LIN {X -0.219,Y -497.782,Z 714.673,A 0.000,B 0.000,C 90.000,E1 337.230} C_DIS
LIN {X 0.009,Y -502.291,Z 714.671,A 0.000,B 0.000,C 90.000,E1 336.794} C_DIS
LIN {X -0.050,Y -508.805,Z 714.668,A 0.000,B 0.000,C 90.000,E1 336.305} C_DIS
LIN {X 0.103,Y -528.863,Z 714.661,A 0.000,B 0.000,C 90.000,E1 334.973} C_DIS
LIN {X -0.127,Y -535.110,Z 714.659,A 0.000,B 0.000,C 90.000,E1 334.588} C_DIS
LIN {X -0.009,Y -541.078,Z 714.656,A 0.000,B 0.000,C 90.000,E1 334.152} C_DIS
LIN {X 0.145,Y -548.131,Z 714.653,A 0.000,B 0.000,C 90.000,E1 333.589} C_DIS
LIN {X -0.065,Y -552.381,Z 714.651,A 0.000,B 0.000,C 90.000,E1 333.256} C_DIS
LIN {X -0.107,Y -557.683,Z 714.649,A 0.000,B 0.000,C 90.000,E1 332.794} C_DIS
LIN {X 0.163,Y -562.857,Z 714.646,A 0.000,B 0.000,C 90.000,E1 332.281} C_DIS
LIN {X 0.153,Y -568.016,Z 714.643,A 0.000,B 0.000,C 90.000,E1 331.769} C_DIS
LIN {X -0.083,Y -574.316,Z 714.640,A 0.000,B 0.000,C 90.000,E1 331.129} C_DIS
LIN {X -0.285,Y -582.771,Z 714.634,A 0.000,B 0.000,C 90.000,E1 330.205} C_DIS
LIN {X -0.328,Y -588.752,Z 714.631,A 0.000,B 0.000,C 90.000,E1 329.537} C_DIS
LIN {X -0.316,Y -594.337,Z 714.627,A 0.000,B 0.000,C 90.000,E1 328.869} C_DIS
LIN {X -0.028,Y -601.884,Z 714.622,A 0.000,B 0.000,C 90.000,E1 327.916} C_DIS
LIN {X 0.100,Y -607.002,Z 714.618,A 0.000,B 0.000,C 90.000,E1 327.248} C_DIS
LIN {X -0.242,Y -611.865,Z 714.615,A 0.000,B 0.000,C 90.000,E1 326.628} C_DIS
LIN {X -0.035,Y -616.443,Z 714.611,A 0.000,B 0.000,C 90.000,E1 325.960} C_DIS
LIN {X 0.030,Y -621.689,Z 714.607,A 0.000,B 0.000,C 90.000,E1 325.182} C_DIS
LIN {X -0.304,Y -628.155,Z 714.601,A 0.000,B 0.000,C 90.000,E1 324.196} C_DIS
LIN {X 0.253,Y -634.206,Z 714.595,A 0.000,B 0.000,C 90.000,E1 323.130} C_DIS
LIN {X -0.001,Y -639.822,Z 714.590,A 0.000,B 0.000,C 90.000,E1 322.145} C_DIS
LIN {X 0.200,Y -644.512,Z 714.585,A 0.000,B 0.000,C 90.000,E1 321.251} C_DIS
LIN {X -0.021,Y -650.301,Z 714.579,A 0.000,B 0.000,C 90.000,E1 320.150} C_DIS
LIN {X 0.256,Y -655.679,Z 714.572,A 0.000,B 0.000,C 90.000,E1 319.013} C_DIS
LIN {X -0.332,Y -660.202,Z 714.567,A 0.000,B 0.000,C 90.000,E1 318.081} C_DIS
LIN {X 0.074,Y -664.376,Z 714.562,A 0.000,B 0.000,C 90.000,E1 317.067} C_DIS
LIN {X 0.054,Y -667.312,Z 714.557,A 0.000,B 0.000,C 90.000,E1 316.338} C_DIS
LIN {X 0.086,Y -670.924,Z 714.552,A 0.000,B 0.000,C 90.000,E1 315.364} C_DIS
LIN {X -0.303,Y -675.162,Z 714.545,A 0.000,B 0.000,C 90.000,E1 314.190} C_DIS
LIN {X -0.155,Y -679.089,Z 714.539,A 0.000,B 0.000,C 90.000,E1 312.975} C_DIS
LIN {X 0.091,Y -682.786,Z 714.532,A 0.000,B 0.000,C 90.000,E1 311.757} C_DIS
LIN {X -0.168,Y -685.479,Z 714.527,A 0.000,B 0.000,C 90.000,E1 310.825} C_DIS
LIN {X 0.124,Y -688.027,Z 714.521,A 0.000,B 0.000,C 90.000,E1 309.850} C_DIS
LIN {X 0.013,Y -690.186,Z 714.516,A 0.000,B 0.000,C 90.000,E1 308.910} C_DIS
LIN {X 0.303,Y -691.640,Z 714.512,A 0.000,B 0.000,C 90.000,E1 308.177} C_DIS
LIN {X 0.247,Y -693.299,Z 714.507,A 0.000,B 0.000,C 90.000,E1 307.237} C_DIS
LIN {X -0.145,Y -695.119,Z 714.500,A 0.000,B 0.000,C 90.000,E1 306.091} C_DIS
LIN {X -0.169,Y -696.354,Z 714.495,A 0.000,B 0.000,C 90.000,E1 305.152} C_DIS
LIN {X -0.353,Y -697.682,Z 714.489,A 0.000,B 0.000,C 90.000,E1 303.992} C_DIS
LIN {X 0.174,Y -698.364,Z 714.485,A 0.000,B 0.000,C 90.000,E1 303.245} C_DIS
LIN {X 0.321,Y -699.714,Z 714.476,A 0.000,B 0.000,C 90.000,E1 301.592} C_DIS
LIN {X 0.166,Y -700.447,Z 714.471,A 0.000,B 0.000,C 90.000,E1 300.669} C_DIS
LIN {X -0.244,Y -700.786,Z 714.467,A 0.000,B 0.000,C 90.000,E1 300.001} C_DIS
LIN {X -0.180,Y -701.290,Z 714.458,A 0.000,B 0.000,C 90.000,E1 298.359} C_DIS
LIN {X -0.160,Y -701.935,Z 714.447,A 0.000,B 0.000,C 90.000,E1 296.488} C_DIS
LIN {X 0.016,Y -702.412,Z 714.442,A 0.000,B 0.000,C 90.000,E1 295.540} C_DIS
LIN {X -0.061,Y -702.510,Z 714.439,A 0.000,B 0.000,C 90.000,E1 295.079} C_DIS
LIN {X 0.201,Y -701.996,Z 714.437,A 0.000,B 0.000,C 90.000,E1 294.591} C_DIS
LIN {X -0.160,Y -701.436,Z 714.435,A 0.000,B 0.000,C 90.000,E1 294.387} C_DIS
LIN {X 0.101,Y -699.381,Z 714.433,A 0.000,B 0.000,C 90.000,E1 293.898} C_DIS
LIN {X 0.237,Y -698.741,Z 714.432,A 0.000,B 0.000,C 90.000,E1 293.770} C_DIS
LIN {X -0.269,Y -697.777,Z 714.432,A 0.000,B 0.000,C 90.000,E1 293.695} C_DIS
LIN {X -0.138,Y -696.354,Z 714.431,A 0.000,B 0.000,C 90.000,E1 293.567} C_DIS
LIN {X 0.001,Y -690.082,Z 714.429,A 0.000,B 0.000,C 90.000,E1 293.153} C_DIS
LIN {X -0.210,Y -687.788,Z 714.428,A 0.000,B 0.000,C 90.000,E1 293.078} C_DIS
LIN {X -0.113,Y -685.753,Z 714.428,A 0.000,B 0.000,C 90.000,E1 293.003} C_DIS
LIN {X -0.153,Y -677.503,Z 714.427,A 0.000,B 0.000,C 90.000,E1 292.823} C_DIS
LIN {X -0.057,Y -659.849,Z 714.426,A 0.000,B 0.000,C 90.000,E1 292.589} C_DIS
LIN {X -0.180,Y -646.131,Z 714.424,A 0.000,B 0.000,C 90.000,E1 292.386} C_DIS
LIN {X -0.277,Y -636.241,Z 714.423,A 0.000,B 0.000,C 90.000,E1 292.206} C_DIS
LIN {X -0.263,Y -622.792,Z 714.422,A 0.000,B 0.000,C 90.000,E1 291.897} C_DIS
LIN {X -0.150,Y -602.290,Z 714.419,A 0.000,B 0.000,C 90.000,E1 291.334} C_DIS
LIN {X 0.095,Y -574.338,Z 714.414,A 0.000,B 0.000,C 90.000,E1 290.482} C_DIS
LIN {X -0.073,Y -567.828,Z 714.413,A 0.000,B 0.000,C 90.000,E1 290.301} C_DIS
LIN {X 0.069,Y -561.417,Z 714.412,A 0.000,B 0.000,C 90.000,E1 290.066} C_DIS
LIN {X -0.026,Y -559.588,Z 714.411,A 0.000,B 0.000,C 90.000,E1 289.993} C_DIS
LIN {X 0.055,Y -556.344,Z 714.410,A 0.000,B 0.000,C 90.000,E1 289.758} C_DIS
LIN {X 0.001,Y -556.275,Z 714.410,A 0.000,B 0.000,C 90.000,E1 289.758} C_DIS
LIN {X -0.250,Y -555.291,Z 714.409,A 0.000,B 0.000,C 90.000,E1 289.577} C_DIS
LIN {X 0.256,Y -554.824,Z 714.407,A 0.000,B 0.000,C 90.000,E1 289.141} C_DIS
LIN {X -0.162,Y -554.077,Z 714.397,A 0.000,B 0.000,C 90.000,E1 287.511} C_DIS
LIN {X -0.230,Y -553.446,Z 714.388,A 0.000,B 0.000,C 90.000,E1 285.843} C_DIS
LIN {X -0.194,Y -552.769,Z 714.377,A 0.000,B 0.000,C 90.000,E1 283.883} C_DIS
LIN {X -0.134,Y -552.316,Z 714.369,A 0.000,B 0.000,C 90.000,E1 282.479} C_DIS
LIN {X -0.075,Y -551.743,Z 714.362,A 0.000,B 0.000,C 90.000,E1 281.074} C_DIS
LIN {X 0.078,Y -550.988,Z 714.352,A 0.000,B 0.000,C 90.000,E1 279.378} C_DIS
LIN {X 0.134,Y -550.123,Z 714.341,A 0.000,B 0.000,C 90.000,E1 277.409} C_DIS
LIN {X 0.270,Y -549.218,Z 714.326,A 0.000,B 0.000,C 90.000,E1 274.588} C_DIS
LIN {X -0.005,Y -548.880,Z 714.318,A 0.000,B 0.000,C 90.000,E1 273.212} C_DIS
LIN {X -0.212,Y -548.201,Z 714.309,A 0.000,B 0.000,C 90.000,E1 271.547} C_DIS
LIN {X 0.029,Y -547.571,Z 714.301,A 0.000,B 0.000,C 90.000,E1 270.115} C_DIS
LIN {X -0.243,Y -546.555,Z 714.291,A 0.000,B 0.000,C 90.000,E1 268.453} C_DIS
LIN {X 0.080,Y -545.356,Z 714.280,A 0.000,B 0.000,C 90.000,E1 266.445} C_DIS
LIN {X -0.226,Y -544.321,Z 714.273,A 0.000,B 0.000,C 90.000,E1 265.065} C_DIS
LIN {X 0.065,Y -543.053,Z 714.263,A 0.000,B 0.000,C 90.000,E1 263.337} C_DIS
LIN {X 0.236,Y -542.050,Z 714.257,A 0.000,B 0.000,C 90.000,E1 262.186} C_DIS
LIN {X 0.077,Y -540.569,Z 714.247,A 0.000,B 0.000,C 90.000,E1 260.500} C_DIS
LIN {X -0.110,Y -539.017,Z 714.238,A 0.000,B 0.000,C 90.000,E1 258.814} C_DIS
LIN {X 0.230,Y -537.809,Z 714.230,A 0.000,B 0.000,C 90.000,E1 257.353} C_DIS
LIN {X -0.268,Y -535.922,Z 714.219,A 0.000,B 0.000,C 90.000,E1 255.408} C_DIS
LIN {X 0.217,Y -534.819,Z 714.212,A 0.000,B 0.000,C 90.000,E1 254.212} C_DIS
LIN {X -0.064,Y -532.775,Z 714.201,A 0.000,B 0.000,C 90.000,E1 252.236} C_DIS
LIN {X 0.061,Y -531.289,Z 714.193,A 0.000,B 0.000,C 90.000,E1 250.786} C_DIS
LIN {X -0.039,Y -529.850,Z 714.187,A 0.000,B 0.000,C 90.000,E1 249.645} C_DIS
LIN {X -0.118,Y -527.448,Z 714.177,A 0.000,B 0.000,C 90.000,E1 247.922} C_DIS
LIN {X -0.215,Y -525.392,Z 714.169,A 0.000,B 0.000,C 90.000,E1 246.485} C_DIS
LIN {X -0.129,Y -523.062,Z 714.161,A 0.000,B 0.000,C 90.000,E1 245.025} C_DIS
LIN {X 0.012,Y -521.122,Z 714.155,A 0.000,B 0.000,C 90.000,E1 243.845} C_DIS
LIN {X 0.112,Y -518.980,Z 714.148,A 0.000,B 0.000,C 90.000,E1 242.666} C_DIS
LIN {X 0.332,Y -515.004,Z 714.137,A 0.000,B 0.000,C 90.000,E1 240.589} C_DIS
LIN {X -0.007,Y -511.908,Z 714.129,A 0.000,B 0.000,C 90.000,E1 239.154} C_DIS
LIN {X 0.022,Y -508.132,Z 714.119,A 0.000,B 0.000,C 90.000,E1 237.375} C_DIS
LIN {X 0.084,Y -505.076,Z 714.111,A 0.000,B 0.000,C 90.000,E1 235.881} C_DIS
LIN {X -0.048,Y -501.706,Z 714.102,A 0.000,B 0.000,C 90.000,E1 234.402} C_DIS
LIN {X 0.005,Y -499.577,Z 714.097,A 0.000,B 0.000,C 90.000,E1 233.497} C_DIS
LIN {X -0.242,Y -498.059,Z 714.094,A 0.000,B 0.000,C 90.000,E1 232.924} C_DIS
LIN {X -0.190,Y -492.612,Z 714.082,A 0.000,B 0.000,C 90.000,E1 230.803} C_DIS
LIN {X 0.028,Y -487.561,Z 714.070,A 0.000,B 0.000,C 90.000,E1 228.647} C_DIS
LIN {X -0.247,Y -484.070,Z 714.062,A 0.000,B 0.000,C 90.000,E1 227.148} C_DIS
LIN {X 0.103,Y -480.666,Z 714.053,A 0.000,B 0.000,C 90.000,E1 225.567} C_DIS
LIN {X -0.063,Y -475.888,Z 714.041,A 0.000,B 0.000,C 90.000,E1 223.419} C_DIS
LIN {X -0.095,Y -471.932,Z 714.031,A 0.000,B 0.000,C 90.000,E1 221.553} C_DIS
LIN {X 0.056,Y -468.580,Z 714.022,A 0.000,B 0.000,C 90.000,E1 219.967} C_DIS
LIN {X 0.135,Y -465.177,Z 714.013,A 0.000,B 0.000,C 90.000,E1 218.382} C_DIS
LIN {X -0.177,Y -459.559,Z 713.999,A 0.000,B 0.000,C 90.000,E1 215.884} C_DIS
LIN {X 0.093,Y -454.588,Z 713.985,A 0.000,B 0.000,C 90.000,E1 213.293} C_DIS
LIN {X 0.197,Y -451.580,Z 713.976,A 0.000,B 0.000,C 90.000,E1 211.671} C_DIS
LIN {X 0.015,Y -448.625,Z 713.967,A 0.000,B 0.000,C 90.000,E1 210.079} C_DIS
LIN {X -0.226,Y -445.600,Z 713.958,A 0.000,B 0.000,C 90.000,E1 208.487} C_DIS
LIN {X 0.047,Y -442.692,Z 713.949,A 0.000,B 0.000,C 90.000,E1 206.821} C_DIS
LIN {X 0.107,Y -439.100,Z 713.938,A 0.000,B 0.000,C 90.000,E1 204.847} C_DIS
LIN {X 0.061,Y -436.090,Z 713.929,A 0.000,B 0.000,C 90.000,E1 203.206} C_DIS
LIN {X 0.049,Y -431.196,Z 713.914,A 0.000,B 0.000,C 90.000,E1 200.556} C_DIS
LIN {X 0.112,Y -428.778,Z 713.907,A 0.000,B 0.000,C 90.000,E1 199.214} C_DIS
LIN {X 0.185,Y -424.473,Z 713.894,A 0.000,B 0.000,C 90.000,E1 196.858} C_DIS
LIN {X -0.111,Y -420.154,Z 713.881,A 0.000,B 0.000,C 90.000,E1 194.537} C_DIS
LIN {X 0.176,Y -415.922,Z 713.867,A 0.000,B 0.000,C 90.000,E1 192.119} C_DIS
LIN {X 0.124,Y -412.367,Z 713.856,A 0.000,B 0.000,C 90.000,E1 190.074} C_DIS
LIN {X -0.083,Y -407.368,Z 713.839,A 0.000,B 0.000,C 90.000,E1 187.004} C_DIS
LIN {X -0.123,Y -404.773,Z 713.829,A 0.000,B 0.000,C 90.000,E1 185.277} C_DIS
LIN {X 0.100,Y -401.334,Z 713.816,A 0.000,B 0.000,C 90.000,E1 182.808} C_DIS
LIN {X 0.032,Y -397.177,Z 713.796,A 0.000,B 0.000,C 90.000,E1 179.312} C_DIS
LIN {X -0.113,Y -394.188,Z 713.779,A 0.000,B 0.000,C 90.000,E1 176.159} C_DIS
LIN {X 0.198,Y -392.236,Z 713.763,A 0.000,B 0.000,C 90.000,E1 173.280} C_DIS
LIN {X -0.130,Y -391.098,Z 713.751,A 0.000,B 0.000,C 90.000,E1 171.197} C_DIS
LIN {X -0.128,Y -389.907,Z 713.733,A 0.000,B 0.000,C 90.000,E1 167.993} C_DIS
LIN {X 0.103,Y -389.112,Z 713.719,A 0.000,B 0.000,C 90.000,E1 165.463} C_DIS
LIN {X 0.064,Y -388.736,Z 713.709,A 0.000,B 0.000,C 90.000,E1 163.685} C_DIS
LIN {X 0.119,Y -388.531,Z 713.700,A 0.000,B 0.000,C 90.000,E1 161.891} C_DIS
LIN {X 0.119,Y -388.413,Z 713.686,A 0.000,B 0.000,C 90.000,E1 159.390} C_DIS
LIN {X 0.101,Y -388.434,Z 713.668,A 0.000,B 0.000,C 90.000,E1 156.177} C_DIS
LIN {X 0.000,Y -388.663,Z 713.654,A 0.000,B 0.000,C 90.000,E1 153.691} C_DIS
LIN {X 0.059,Y -388.912,Z 713.644,A 0.000,B 0.000,C 90.000,E1 151.897} C_DIS
LIN {X 0.061,Y -389.865,Z 713.624,A 0.000,B 0.000,C 90.000,E1 148.329} C_DIS
LIN {X 0.145,Y -393.306,Z 713.596,A 0.000,B 0.000,C 90.000,E1 143.336} C_DIS
LIN {X -0.120,Y -395.537,Z 713.585,A 0.000,B 0.000,C 90.000,E1 141.251} C_DIS
LIN {X 0.067,Y -399.294,Z 713.569,A 0.000,B 0.000,C 90.000,E1 138.405} C_DIS
LIN {X -0.206,Y -401.196,Z 713.563,A 0.000,B 0.000,C 90.000,E1 137.391} C_DIS
LIN {X 0.178,Y -402.104,Z 713.561,A 0.000,B 0.000,C 90.000,E1 136.986} C_DIS
LIN {X -0.061,Y -403.913,Z 713.558,A 0.000,B 0.000,C 90.000,E1 136.458} C_DIS
LIN {X 0.254,Y -406.545,Z 713.555,A 0.000,B 0.000,C 90.000,E1 135.891} C_DIS
LIN {X 0.062,Y -410.220,Z 713.552,A 0.000,B 0.000,C 90.000,E1 135.405} C_DIS
LIN {X -0.051,Y -414.965,Z 713.549,A 0.000,B 0.000,C 90.000,E1 134.879} C_DIS
LIN {X 0.100,Y -431.494,Z 713.540,A 0.000,B 0.000,C 90.000,E1 133.218} C_DIS
LIN {X -0.272,Y -446.498,Z 713.533,A 0.000,B 0.000,C 90.000,E1 131.919} C_DIS
LIN {X 0.289,Y -461.223,Z 713.525,A 0.000,B 0.000,C 90.000,E1 130.539} C_DIS
LIN {X 0.262,Y -467.053,Z 713.523,A 0.000,B 0.000,C 90.000,E1 130.011} C_DIS
LIN {X -0.259,Y -475.583,Z 713.518,A 0.000,B 0.000,C 90.000,E1 129.277} C_DIS
LIN {X -0.252,Y -483.867,Z 713.514,A 0.000,B 0.000,C 90.000,E1 128.463} C_DIS
LIN {X 0.009,Y -490.789,Z 713.510,A 0.000,B 0.000,C 90.000,E1 127.729} C_DIS
LIN {X 0.138,Y -498.849,Z 713.505,A 0.000,B 0.000,C 90.000,E1 126.870} C_DIS
LIN {X 0.003,Y -503.973,Z 713.502,A 0.000,B 0.000,C 90.000,E1 126.297} C_DIS
LIN {X 0.113,Y -508.637,Z 713.499,A 0.000,B 0.000,C 90.000,E1 125.724} C_DIS
LIN {X 0.136,Y -511.959,Z 713.496,A 0.000,B 0.000,C 90.000,E1 125.311} C_DIS
LIN {X 0.009,Y -516.326,Z 713.493,A 0.000,B 0.000,C 90.000,E1 124.739} C_DIS
LIN {X -0.022,Y -521.127,Z 713.489,A 0.000,B 0.000,C 90.000,E1 124.040} C_DIS
LIN {X 0.053,Y -524.742,Z 713.486,A 0.000,B 0.000,C 90.000,E1 123.452} C_DIS
LIN {X -0.191,Y -528.871,Z 713.482,A 0.000,B 0.000,C 90.000,E1 122.752} C_DIS
LIN {X 0.047,Y -532.656,Z 713.478,A 0.000,B 0.000,C 90.000,E1 122.005} C_DIS
LIN {X 0.318,Y -536.161,Z 713.474,A 0.000,B 0.000,C 90.000,E1 121.258} C_DIS
LIN {X -0.115,Y -539.405,Z 713.470,A 0.000,B 0.000,C 90.000,E1 120.590} C_DIS
LIN {X 0.160,Y -544.830,Z 713.463,A 0.000,B 0.000,C 90.000,E1 119.283} C_DIS
LIN {X 0.149,Y -548.288,Z 713.458,A 0.000,B 0.000,C 90.000,E1 118.437} C_DIS
LIN {X 0.172,Y -551.514,Z 713.453,A 0.000,B 0.000,C 90.000,E1 117.590} C_DIS
LIN {X 0.006,Y -555.477,Z 713.447,A 0.000,B 0.000,C 90.000,E1 116.488} C_DIS
LIN {X -0.146,Y -558.163,Z 713.443,A 0.000,B 0.000,C 90.000,E1 115.668} C_DIS
LIN {X -0.030,Y -560.624,Z 713.438,A 0.000,B 0.000,C 90.000,E1 114.823} C_DIS
LIN {X -0.132,Y -562.734,Z 713.433,A 0.000,B 0.000,C 90.000,E1 114.003} C_DIS
LIN {X 0.083,Y -564.618,Z 713.429,A 0.000,B 0.000,C 90.000,E1 113.153} C_DIS
LIN {X 0.025,Y -566.225,Z 713.424,A 0.000,B 0.000,C 90.000,E1 112.333} C_DIS
LIN {X 0.256,Y -569.035,Z 713.415,A 0.000,B 0.000,C 90.000,E1 110.663} C_DIS
LIN {X 0.151,Y -571.704,Z 713.406,A 0.000,B 0.000,C 90.000,E1 109.033} C_DIS
LIN {X 0.119,Y -573.403,Z 713.400,A 0.000,B 0.000,C 90.000,E1 107.946} C_DIS
LIN {X -0.252,Y -576.205,Z 713.389,A 0.000,B 0.000,C 90.000,E1 106.079} C_DIS
LIN {X 0.026,Y -578.470,Z 713.380,A 0.000,B 0.000,C 90.000,E1 104.426} C_DIS
LIN {X 0.135,Y -580.319,Z 713.373,A 0.000,B 0.000,C 90.000,E1 103.063} C_DIS
LIN {X -0.196,Y -582.549,Z 713.364,A 0.000,B 0.000,C 90.000,E1 101.478} C_DIS
LIN {X 0.175,Y -584.057,Z 713.358,A 0.000,B 0.000,C 90.000,E1 100.366} C_DIS
LIN {X 0.219,Y -585.156,Z 713.353,A 0.000,B 0.000,C 90.000,E1 99.557} C_DIS
LIN {X -0.226,Y -587.055,Z 713.344,A 0.000,B 0.000,C 90.000,E1 97.992} C_DIS
LIN {X -0.304,Y -588.577,Z 713.337,A 0.000,B 0.000,C 90.000,E1 96.663} C_DIS
LIN {X -0.024,Y -589.717,Z 713.331,A 0.000,B 0.000,C 90.000,E1 95.568} C_DIS
LIN {X 0.124,Y -591.401,Z 713.322,A 0.000,B 0.000,C 90.000,E1 93.955} C_DIS
LIN {X -0.198,Y -592.398,Z 713.316,A 0.000,B 0.000,C 90.000,E1 92.922} C_DIS
LIN {X 0.297,Y -593.492,Z 713.309,A 0.000,B 0.000,C 90.000,E1 91.547} C_DIS
LIN {X -0.167,Y -594.566,Z 713.300,A 0.000,B 0.000,C 90.000,E1 90.000} C_DIS
LIN {X 0.131,Y -595.069,Z 713.294,A 0.000,B 0.000,C 90.000,E1 88.912} C_DIS
LIN {X 0.080,Y -595.558,Z 713.287,A 0.000,B 0.000,C 90.000,E1 87.593} C_DIS
LIN {X 0.039,Y -595.887,Z 713.279,A 0.000,B 0.000,C 90.000,E1 86.274} C_DIS
LIN {X -0.227,Y -596.071,Z 713.273,A 0.000,B 0.000,C 90.000,E1 85.241} C_DIS
LIN {X -0.166,Y -596.122,Z 713.266,A 0.000,B 0.000,C 90.000,E1 83.913} C_DIS
LIN {X -0.166,Y -596.057,Z 713.259,A 0.000,B 0.000,C 90.000,E1 82.591} C_DIS
LIN {X 0.290,Y -595.889,Z 713.253,A 0.000,B 0.000,C 90.000,E1 81.489} C_DIS
LIN {X -0.142,Y -595.376,Z 713.246,A 0.000,B 0.000,C 90.000,E1 80.208} C_DIS
LIN {X -0.277,Y -594.837,Z 713.240,A 0.000,B 0.000,C 90.000,E1 79.162} C_DIS
LIN {X 0.257,Y -593.802,Z 713.231,A 0.000,B 0.000,C 90.000,E1 77.521} C_DIS
LIN {X -0.089,Y -592.801,Z 713.224,A 0.000,B 0.000,C 90.000,E1 76.228} C_DIS
LIN {X -0.155,Y -591.870,Z 713.218,A 0.000,B 0.000,C 90.000,E1 75.172} C_DIS
LIN {X 0.335,Y -590.664,Z 713.210,A 0.000,B 0.000,C 90.000,E1 73.795} C_DIS
LIN {X 0.069,Y -589.317,Z 713.203,A 0.000,B 0.000,C 90.000,E1 72.489} C_DIS
LIN {X -0.287,Y -588.117,Z 713.197,A 0.000,B 0.000,C 90.000,E1 71.456} C_DIS
LIN {X -0.012,Y -586.188,Z 713.188,A 0.000,B 0.000,C 90.000,E1 69.826} C_DIS
LIN {X 0.211,Y -584.312,Z 713.181,A 0.000,B 0.000,C 90.000,E1 68.465} C_DIS
LIN {X 0.137,Y -583.098,Z 713.176,A 0.000,B 0.000,C 90.000,E1 67.667} C_DIS
LIN {X -0.227,Y -580.812,Z 713.169,A 0.000,B 0.000,C 90.000,E1 66.357} C_DIS
LIN {X 0.278,Y -578.645,Z 713.163,A 0.000,B 0.000,C 90.000,E1 65.229} C_DIS
LIN {X -0.150,Y -576.866,Z 713.158,A 0.000,B 0.000,C 90.000,E1 64.460} C_DIS
LIN {X -0.227,Y -574.275,Z 713.152,A 0.000,B 0.000,C 90.000,E1 63.384} C_DIS
LIN {X 0.076,Y -572.115,Z 713.148,A 0.000,B 0.000,C 90.000,E1 62.538} C_DIS
LIN {X 0.188,Y -568.886,Z 713.141,A 0.000,B 0.000,C 90.000,E1 61.435} C_DIS
LIN {X -0.060,Y -566.330,Z 713.137,A 0.000,B 0.000,C 90.000,E1 60.639} C_DIS
LIN {X 0.156,Y -563.484,Z 713.132,A 0.000,B 0.000,C 90.000,E1 59.793} C_DIS
LIN {X 0.053,Y -561.491,Z 713.129,A 0.000,B 0.000,C 90.000,E1 59.253} C_DIS
LIN {X 0.205,Y -558.178,Z 713.125,A 0.000,B 0.000,C 90.000,E1 58.408} C_DIS
LIN {X -0.048,Y -555.191,Z 713.121,A 0.000,B 0.000,C 90.000,E1 57.740} C_DIS
LIN {X -0.031,Y -551.798,Z 713.117,A 0.000,B 0.000,C 90.000,E1 57.041} C_DIS
LIN {X -0.041,Y -547.985,Z 713.113,A 0.000,B 0.000,C 90.000,E1 56.342} C_DIS
LIN {X -0.080,Y -543.761,Z 713.109,A 0.000,B 0.000,C 90.000,E1 55.642} C_DIS
LIN {X 0.149,Y -540.240,Z 713.106,A 0.000,B 0.000,C 90.000,E1 55.055} C_DIS
LIN {X 0.185,Y -536.382,Z 713.103,A 0.000,B 0.000,C 90.000,E1 54.482} C_DIS
LIN {X 0.194,Y -532.078,Z 713.100,A 0.000,B 0.000,C 90.000,E1 53.909} C_DIS
LIN {X 0.174,Y -527.262,Z 713.096,A 0.000,B 0.000,C 90.000,E1 53.336} C_DIS
LIN {X -0.230,Y -522.297,Z 713.094,A 0.000,B 0.000,C 90.000,E1 52.844} C_DIS
LIN {X 0.003,Y -517.101,Z 713.091,A 0.000,B 0.000,C 90.000,E1 52.316} C_DIS
LIN {X 0.150,Y -512.572,Z 713.089,A 0.000,B 0.000,C 90.000,E1 51.904} C_DIS
LIN {X -0.134,Y -506.355,Z 713.086,A 0.000,B 0.000,C 90.000,E1 51.457} C_DIS
LIN {X 0.068,Y -501.512,Z 713.084,A 0.000,B 0.000,C 90.000,E1 51.090} C_DIS
LIN {X 0.093,Y -493.549,Z 713.081,A 0.000,B 0.000,C 90.000,E1 50.561} C_DIS
LIN {X -0.121,Y -488.562,Z 713.079,A 0.000,B 0.000,C 90.000,E1 50.275} C_DIS
LIN {X -0.156,Y -472.147,Z 713.074,A 0.000,B 0.000,C 90.000,E1 49.299} C_DIS
LIN {X 0.138,Y -452.641,Z 713.067,A 0.000,B 0.000,C 90.000,E1 48.081} C_DIS
LIN {X -0.132,Y -427.469,Z 713.058,A 0.000,B 0.000,C 90.000,E1 46.458} C_DIS
LIN {X -0.227,Y -422.791,Z 713.056,A 0.000,B 0.000,C 90.000,E1 46.134} C_DIS
LIN {X -0.283,Y -420.646,Z 713.055,A 0.000,B 0.000,C 90.000,E1 45.972} C_DIS
LIN {X 0.283,Y -420.618,Z 713.055,A 0.000,B 0.000,C 90.000,E1 45.891} C_DIS
LIN {X 0.031,Y -418.406,Z 713.049,A 0.000,B 0.000,C 90.000,E1 44.717} C_DIS
LIN {X 0.137,Y -408.883,Z 713.024,A 0.000,B 0.000,C 90.000,E1 40.253} C_DIS
LIN {X -0.101,Y -407.965,Z 713.021,A 0.000,B 0.000,C 90.000,E1 39.769} C_DIS
LIN {X 0.132,Y -407.809,Z 713.020,A 0.000,B 0.000,C 90.000,E1 39.564} C_DIS
LIN {X 0.059,Y -408.275,Z 713.000,A 0.000,B 0.000,C 90.000,E1 35.931} C_DIS
LIN {X 0.003,Y -409.059,Z 712.988,A 0.000,B 0.000,C 90.000,E1 33.865} C_DIS
LIN {X -0.031,Y -409.988,Z 712.977,A 0.000,B 0.000,C 90.000,E1 31.799} C_DIS
LIN {X 0.086,Y -411.406,Z 712.961,A 0.000,B 0.000,C 90.000,E1 29.027} C_DIS
LIN {X 0.119,Y -412.824,Z 712.948,A 0.000,B 0.000,C 90.000,E1 26.616} C_DIS
LIN {X -0.058,Y -414.831,Z 712.933,A 0.000,B 0.000,C 90.000,E1 23.898} C_DIS
LIN {X 0.188,Y -417.555,Z 712.916,A 0.000,B 0.000,C 90.000,E1 20.791} C_DIS
LIN {X 0.137,Y -420.036,Z 712.902,A 0.000,B 0.000,C 90.000,E1 18.417} C_DIS
LIN {X 0.064,Y -422.009,Z 712.893,A 0.000,B 0.000,C 90.000,E1 16.732} C_DIS
LIN {X 0.160,Y -424.959,Z 712.880,A 0.000,B 0.000,C 90.000,E1 14.356} C_DIS
LIN {X 0.042,Y -427.653,Z 712.869,A 0.000,B 0.000,C 90.000,E1 12.355} C_DIS
LIN {X 0.210,Y -429.901,Z 712.859,A 0.000,B 0.000,C 90.000,E1 10.658} C_DIS
LIN {X 0.035,Y -432.694,Z 712.848,A 0.000,B 0.000,C 90.000,E1 8.681} C_DIS
LIN {X 0.101,Y -435.054,Z 712.839,A 0.000,B 0.000,C 90.000,E1 7.011} C_DIS
LIN {X -0.164,Y -437.478,Z 712.830,A 0.000,B 0.000,C 90.000,E1 5.391} C_DIS
LIN {X -0.116,Y -441.574,Z 712.815,A 0.000,B 0.000,C 90.000,E1 2.751} C_DIS
LIN {X 0.206,Y -444.939,Z 712.804,A 0.000,B 0.000,C 90.000,E1 0.745} C_DIS
LIN {X 0.157,Y -448.557,Z 712.793,A 0.000,B 0.000,C 90.000,E1 358.797} C_DIS
LIN {X 0.040,Y -451.675,Z 712.784,A 0.000,B 0.000,C 90.000,E1 357.192} C_DIS
LIN {X 0.176,Y -455.591,Z 712.774,A 0.000,B 0.000,C 90.000,E1 355.241} C_DIS
LIN {X 0.032,Y -459.564,Z 712.763,A 0.000,B 0.000,C 90.000,E1 353.337} C_DIS
LIN {X 0.013,Y -462.233,Z 712.756,A 0.000,B 0.000,C 90.000,E1 352.064} C_DIS
LIN {X 0.092,Y -465.973,Z 712.745,A 0.000,B 0.000,C 90.000,E1 350.151} C_DIS
LIN {X 0.244,Y -468.431,Z 712.738,A 0.000,B 0.000,C 90.000,E1 348.870} C_DIS
LIN {X -0.030,Y -470.763,Z 712.731,A 0.000,B 0.000,C 90.000,E1 347.645} C_DIS
LIN {X 0.056,Y -474.151,Z 712.721,A 0.000,B 0.000,C 90.000,E1 345.755} C_DIS
LIN {X -0.037,Y -476.479,Z 712.714,A 0.000,B 0.000,C 90.000,E1 344.519} C_DIS
LIN {X 0.107,Y -481.862,Z 712.698,A 0.000,B 0.000,C 90.000,E1 341.710} C_DIS
LIN {X -0.024,Y -487.150,Z 712.685,A 0.000,B 0.000,C 90.000,E1 339.263} C_DIS
LIN {X 0.014,Y -488.813,Z 712.681,A 0.000,B 0.000,C 90.000,E1 338.646} C_DIS
LIN {X 0.039,Y -489.793,Z 712.680,A 0.000,B 0.000,C 90.000,E1 338.337} C_DIS
LIN {X -0.128,Y -491.618,Z 712.677,A 0.000,B 0.000,C 90.000,E1 337.901} C_DIS
LIN {X 0.134,Y -492.299,Z 712.676,A 0.000,B 0.000,C 90.000,E1 337.720} C_DIS
LIN {X -0.033,Y -495.392,Z 712.674,A 0.000,B 0.000,C 90.000,E1 337.283} C_DIS
LIN {X 0.218,Y -496.793,Z 712.673,A 0.000,B 0.000,C 90.000,E1 337.102} C_DIS
LIN {X 0.030,Y -499.743,Z 712.671,A 0.000,B 0.000,C 90.000,E1 336.847} C_DIS
LIN {X 0.114,Y -502.431,Z 712.670,A 0.000,B 0.000,C 90.000,E1 336.561} C_DIS
LIN {X 0.050,Y -506.680,Z 712.668,A 0.000,B 0.000,C 90.000,E1 336.230} C_DIS
LIN {X -0.110,Y -525.677,Z 712.661,A 0.000,B 0.000,C 90.000,E1 334.973} C_DIS
LIN {X -0.062,Y -533.493,Z 712.658,A 0.000,B 0.000,C 90.000,E1 334.460} C_DIS
LIN {X 0.281,Y -540.988,Z 712.655,A 0.000,B 0.000,C 90.000,E1 333.896} C_DIS
LIN {X 0.184,Y -546.773,Z 712.653,A 0.000,B 0.000,C 90.000,E1 333.461} C_DIS
LIN {X 0.099,Y -552.502,Z 712.650,A 0.000,B 0.000,C 90.000,E1 332.999} C_DIS
LIN {X -0.124,Y -557.963,Z 712.647,A 0.000,B 0.000,C 90.000,E1 332.538} C_DIS
LIN {X -0.060,Y -564.657,Z 712.644,A 0.000,B 0.000,C 90.000,E1 331.897} C_DIS
LIN {X -0.201,Y -571.073,Z 712.640,A 0.000,B 0.000,C 90.000,E1 331.257} C_DIS
LIN {X -0.207,Y -577.222,Z 712.637,A 0.000,B 0.000,C 90.000,E1 330.589} C_DIS
LIN {X -0.179,Y -584.333,Z 712.632,A 0.000,B 0.000,C 90.000,E1 329.793} C_DIS
LIN {X -0.133,Y -589.074,Z 712.629,A 0.000,B 0.000,C 90.000,E1 329.253} C_DIS
LIN {X -0.267,Y -597.994,Z 712.623,A 0.000,B 0.000,C 90.000,E1 328.201} C_DIS
LIN {X 0.106,Y -604.366,Z 712.619,A 0.000,B 0.000,C 90.000,E1 327.375} C_DIS
LIN {X -0.288,Y -610.333,Z 712.615,A 0.000,B 0.000,C 90.000,E1 326.628} C_DIS
LIN {X 0.224,Y -615.935,Z 712.610,A 0.000,B 0.000,C 90.000,E1 325.801} C_DIS
LIN {X -0.046,Y -620.376,Z 712.607,A 0.000,B 0.000,C 90.000,E1 325.182} C_DIS
LIN {X 0.098,Y -626.940,Z 712.601,A 0.000,B 0.000,C 90.000,E1 324.149} C_DIS
LIN {X 0.130,Y -633.104,Z 712.595,A 0.000,B 0.000,C 90.000,E1 323.130} C_DIS
LIN {X 0.252,Y -638.807,Z 712.590,A 0.000,B 0.000,C 90.000,E1 322.110} C_DIS
LIN {X -0.042,Y -644.888,Z 712.583,A 0.000,B 0.000,C 90.000,E1 321.009} C_DIS
LIN {X 0.236,Y -650.077,Z 712.578,A 0.000,B 0.000,C 90.000,E1 319.989} C_DIS
LIN {X 0.068,Y -654.343,Z 712.573,A 0.000,B 0.000,C 90.000,E1 319.138} C_DIS
LIN {X -0.039,Y -658.965,Z 712.568,A 0.000,B 0.000,C 90.000,E1 318.162} C_DIS
LIN {X 0.351,Y -663.259,Z 712.562,A 0.000,B 0.000,C 90.000,E1 317.148} C_DIS
LIN {X -0.143,Y -667.244,Z 712.557,A 0.000,B 0.000,C 90.000,E1 316.215} C_DIS
LIN {X -0.127,Y -670.891,Z 712.551,A 0.000,B 0.000,C 90.000,E1 315.243} C_DIS
LIN {X -0.038,Y -675.159,Z 712.545,A 0.000,B 0.000,C 90.000,E1 314.028} C_DIS
LIN {X -0.353,Y -679.114,Z 712.538,A 0.000,B 0.000,C 90.000,E1 312.852} C_DIS
LIN {X 0.356,Y -682.886,Z 712.531,A 0.000,B 0.000,C 90.000,E1 311.595} C_DIS
LIN {X -0.298,Y -686.276,Z 712.525,A 0.000,B 0.000,C 90.000,E1 310.458} C_DIS
LIN {X -0.051,Y -688.155,Z 712.521,A 0.000,B 0.000,C 90.000,E1 309.725} C_DIS
LIN {X 0.278,Y -690.306,Z 712.515,A 0.000,B 0.000,C 90.000,E1 308.749} C_DIS
LIN {X -0.403,Y -691.763,Z 712.512,A 0.000,B 0.000,C 90.000,E1 308.096} C_DIS
LIN {X 0.091,Y -693.432,Z 712.506,A 0.000,B 0.000,C 90.000,E1 307.111} C_DIS
LIN {X 0.115,Y -695.263,Z 712.500,A 0.000,B 0.000,C 90.000,E1 305.931} C_DIS
LIN {X -0.313,Y -696.504,Z 712.495,A 0.000,B 0.000,C 90.000,E1 305.025} C_DIS
LIN {X -0.101,Y -697.838,Z 712.488,A 0.000,B 0.000,C 90.000,E1 303.833} C_DIS
LIN {X 0.423,Y -698.516,Z 712.484,A 0.000,B 0.000,C 90.000,E1 303.086} C_DIS
LIN {X 0.195,Y -699.902,Z 712.475,A 0.000,B 0.000,C 90.000,E1 301.465} C_DIS
LIN {X 0.044,Y -700.609,Z 712.470,A 0.000,B 0.000,C 90.000,E1 300.541} C_DIS
LIN {X -0.363,Y -700.896,Z 712.466,A 0.000,B 0.000,C 90.000,E1 299.873} C_DIS
LIN {X 0.048,Y -701.328,Z 712.458,A 0.000,B 0.000,C 90.000,E1 298.437} C_DIS
LIN {X 0.116,Y -701.873,Z 712.449,A 0.000,B 0.000,C 90.000,E1 296.796} C_DIS
LIN {X -0.092,Y -702.570,Z 712.441,A 0.000,B 0.000,C 90.000,E1 295.412} C_DIS
LIN {X 0.187,Y -702.648,Z 712.440,A 0.000,B 0.000,C 90.000,E1 295.155} C_DIS
LIN {X -0.186,Y -702.179,Z 712.437,A 0.000,B 0.000,C 90.000,E1 294.719} C_DIS
LIN {X 0.094,Y -701.832,Z 712.436,A 0.000,B 0.000,C 90.000,E1 294.463} C_DIS
LIN {X 0.004,Y -699.843,Z 712.433,A 0.000,B 0.000,C 90.000,E1 294.003} C_DIS
LIN {X -0.010,Y -698.522,Z 712.432,A 0.000,B 0.000,C 90.000,E1 293.770} C_DIS
LIN {X 0.123,Y -697.480,Z 712.431,A 0.000,B 0.000,C 90.000,E1 293.643} C_DIS
LIN {X 0.254,Y -695.913,Z 712.431,A 0.000,B 0.000,C 90.000,E1 293.515} C_DIS
LIN {X -0.238,Y -691.236,Z 712.429,A 0.000,B 0.000,C 90.000,E1 293.259} C_DIS
LIN {X 0.189,Y -689.594,Z 712.429,A 0.000,B 0.000,C 90.000,E1 293.131} C_DIS
LIN {X -0.210,Y -687.350,Z 712.428,A 0.000,B 0.000,C 90.000,E1 293.078} C_DIS
LIN {X 0.291,Y -684.141,Z 712.428,A 0.000,B 0.000,C 90.000,E1 292.950} C_DIS
LIN {X 0.225,Y -678.075,Z 712.427,A 0.000,B 0.000,C 90.000,E1 292.823} C_DIS
LIN {X -0.321,Y -656.752,Z 712.425,A 0.000,B 0.000,C 90.000,E1 292.589} C_DIS
LIN {X 0.128,Y -646.475,Z 712.424,A 0.000,B 0.000,C 90.000,E1 292.386} C_DIS
LIN {X 0.048,Y -636.631,Z 712.423,A 0.000,B 0.000,C 90.000,E1 292.206} C_DIS
LIN {X 0.068,Y -623.177,Z 712.422,A 0.000,B 0.000,C 90.000,E1 291.897} C_DIS
LIN {X -0.036,Y -602.662,Z 712.419,A 0.000,B 0.000,C 90.000,E1 291.354} C_DIS
LIN {X 0.162,Y -578.280,Z 712.415,A 0.000,B 0.000,C 90.000,E1 290.610} C_DIS
LIN {X 0.059,Y -567.806,Z 712.413,A 0.000,B 0.000,C 90.000,E1 290.301} C_DIS
LIN {X 0.198,Y -561.447,Z 712.412,A 0.000,B 0.000,C 90.000,E1 290.066} C_DIS
LIN {X 0.102,Y -559.605,Z 712.411,A 0.000,B 0.000,C 90.000,E1 289.993} C_DIS
LIN {X 0.067,Y -556.201,Z 712.410,A 0.000,B 0.000,C 90.000,E1 289.758} C_DIS
LIN {X 0.035,Y -556.169,Z 712.410,A 0.000,B 0.000,C 90.000,E1 289.758} C_DIS
LIN {X -0.070,Y -555.273,Z 712.409,A 0.000,B 0.000,C 90.000,E1 289.577} C_DIS
LIN {X 0.100,Y -554.766,Z 712.406,A 0.000,B 0.000,C 90.000,E1 289.141} C_DIS
LIN {X 0.208,Y -554.040,Z 712.397,A 0.000,B 0.000,C 90.000,E1 287.457} C_DIS
LIN {X 0.145,Y -553.409,Z 712.388,A 0.000,B 0.000,C 90.000,E1 285.788} C_DIS
LIN {X 0.065,Y -552.828,Z 712.379,A 0.000,B 0.000,C 90.000,E1 284.120} C_DIS
LIN {X -0.294,Y -552.247,Z 712.369,A 0.000,B 0.000,C 90.000,E1 282.479} C_DIS
LIN {X 0.294,Y -551.824,Z 712.363,A 0.000,B 0.000,C 90.000,E1 281.299} C_DIS
LIN {X -0.197,Y -551.044,Z 712.354,A 0.000,B 0.000,C 90.000,E1 279.670} C_DIS
LIN {X -0.134,Y -550.186,Z 712.343,A 0.000,B 0.000,C 90.000,E1 277.701} C_DIS
LIN {X -0.027,Y -549.316,Z 712.329,A 0.000,B 0.000,C 90.000,E1 275.163} C_DIS
LIN {X -0.264,Y -549.036,Z 712.321,A 0.000,B 0.000,C 90.000,E1 273.784} C_DIS
LIN {X -0.043,Y -548.639,Z 712.315,A 0.000,B 0.000,C 90.000,E1 272.636} C_DIS
LIN {X 0.220,Y -548.137,Z 712.307,A 0.000,B 0.000,C 90.000,E1 271.203} C_DIS
LIN {X -0.133,Y -547.626,Z 712.301,A 0.000,B 0.000,C 90.000,E1 270.115} C_DIS
LIN {X 0.201,Y -546.403,Z 712.290,A 0.000,B 0.000,C 90.000,E1 268.108} C_DIS
LIN {X -0.118,Y -545.588,Z 712.282,A 0.000,B 0.000,C 90.000,E1 266.731} C_DIS
LIN {X 0.083,Y -544.568,Z 712.274,A 0.000,B 0.000,C 90.000,E1 265.298} C_DIS
LIN {X -0.171,Y -543.307,Z 712.265,A 0.000,B 0.000,C 90.000,E1 263.628} C_DIS
LIN {X 0.072,Y -542.341,Z 712.258,A 0.000,B 0.000,C 90.000,E1 262.470} C_DIS
LIN {X -0.157,Y -540.837,Z 712.249,A 0.000,B 0.000,C 90.000,E1 260.792} C_DIS
LIN {X 0.121,Y -539.554,Z 712.241,A 0.000,B 0.000,C 90.000,E1 259.342} C_DIS
LIN {X 0.074,Y -537.794,Z 712.230,A 0.000,B 0.000,C 90.000,E1 257.353} C_DIS
LIN {X 0.094,Y -535.907,Z 712.219,A 0.000,B 0.000,C 90.000,E1 255.353} C_DIS
LIN {X 0.061,Y -534.804,Z 712.212,A 0.000,B 0.000,C 90.000,E1 254.212} C_DIS
LIN {X 0.095,Y -533.071,Z 712.203,A 0.000,B 0.000,C 90.000,E1 252.489} C_DIS
LIN {X 0.216,Y -531.612,Z 712.195,A 0.000,B 0.000,C 90.000,E1 251.040} C_DIS
LIN {X -0.199,Y -530.226,Z 712.188,A 0.000,B 0.000,C 90.000,E1 249.934} C_DIS
LIN {X 0.052,Y -528.274,Z 712.180,A 0.000,B 0.000,C 90.000,E1 248.465} C_DIS
LIN {X 0.082,Y -526.649,Z 712.174,A 0.000,B 0.000,C 90.000,E1 247.305} C_DIS
LIN {X -0.199,Y -524.964,Z 712.168,A 0.000,B 0.000,C 90.000,E1 246.177} C_DIS
LIN {X 0.031,Y -522.091,Z 712.158,A 0.000,B 0.000,C 90.000,E1 244.409} C_DIS
LIN {X -0.089,Y -520.082,Z 712.151,A 0.000,B 0.000,C 90.000,E1 243.256} C_DIS
LIN {X -0.238,Y -517.810,Z 712.145,A 0.000,B 0.000,C 90.000,E1 242.103} C_DIS
LIN {X 0.182,Y -514.974,Z 712.137,A 0.000,B 0.000,C 90.000,E1 240.589} C_DIS
LIN {X 0.106,Y -511.874,Z 712.129,A 0.000,B 0.000,C 90.000,E1 239.125} C_DIS
LIN {X -0.127,Y -508.096,Z 712.119,A 0.000,B 0.000,C 90.000,E1 237.375} C_DIS
LIN {X -0.066,Y -505.010,Z 712.110,A 0.000,B 0.000,C 90.000,E1 235.881} C_DIS
LIN {X -0.198,Y -501.679,Z 712.102,A 0.000,B 0.000,C 90.000,E1 234.402} C_DIS
LIN {X -0.144,Y -499.539,Z 712.097,A 0.000,B 0.000,C 90.000,E1 233.497} C_DIS
LIN {X 0.049,Y -496.446,Z 712.090,A 0.000,B 0.000,C 90.000,E1 232.271} C_DIS
LIN {X 0.057,Y -489.666,Z 712.075,A 0.000,B 0.000,C 90.000,E1 229.542} C_DIS
LIN {X 0.182,Y -486.100,Z 712.067,A 0.000,B 0.000,C 90.000,E1 228.000} C_DIS
LIN {X 0.237,Y -482.635,Z 712.058,A 0.000,B 0.000,C 90.000,E1 226.458} C_DIS
LIN {X -0.044,Y -480.616,Z 712.053,A 0.000,B 0.000,C 90.000,E1 225.567} C_DIS
LIN {X 0.118,Y -475.845,Z 712.041,A 0.000,B 0.000,C 90.000,E1 223.380} C_DIS
LIN {X 0.072,Y -471.832,Z 712.031,A 0.000,B 0.000,C 90.000,E1 221.515} C_DIS
LIN {X 0.211,Y -468.477,Z 712.022,A 0.000,B 0.000,C 90.000,E1 219.930} C_DIS
LIN {X -0.013,Y -465.087,Z 712.013,A 0.000,B 0.000,C 90.000,E1 218.382} C_DIS
LIN {X -0.054,Y -459.519,Z 711.999,A 0.000,B 0.000,C 90.000,E1 215.851} C_DIS
LIN {X 0.222,Y -455.171,Z 711.987,A 0.000,B 0.000,C 90.000,E1 213.579} C_DIS
LIN {X -0.042,Y -452.164,Z 711.978,A 0.000,B 0.000,C 90.000,E1 212.005} C_DIS
LIN {X -0.053,Y -447.983,Z 711.965,A 0.000,B 0.000,C 90.000,E1 209.745} C_DIS
LIN {X -0.004,Y -443.844,Z 711.953,A 0.000,B 0.000,C 90.000,E1 207.462} C_DIS
LIN {X -0.160,Y -440.839,Z 711.944,A 0.000,B 0.000,C 90.000,E1 205.848} C_DIS
LIN {X -0.172,Y -437.851,Z 711.934,A 0.000,B 0.000,C 90.000,E1 204.207} C_DIS
LIN {X -0.249,Y -435.400,Z 711.927,A 0.000,B 0.000,C 90.000,E1 202.898} C_DIS
LIN {X 0.086,Y -431.762,Z 711.916,A 0.000,B 0.000,C 90.000,E1 200.865} C_DIS
LIN {X -0.246,Y -429.369,Z 711.909,A 0.000,B 0.000,C 90.000,E1 199.577} C_DIS
LIN {X 0.184,Y -425.678,Z 711.897,A 0.000,B 0.000,C 90.000,E1 197.511} C_DIS
LIN {X 0.079,Y -422.591,Z 711.888,A 0.000,B 0.000,C 90.000,E1 195.843} C_DIS
LIN {X -0.026,Y -418.924,Z 711.877,A 0.000,B 0.000,C 90.000,E1 193.828} C_DIS
LIN {X 0.136,Y -414.738,Z 711.864,A 0.000,B 0.000,C 90.000,E1 191.422} C_DIS
LIN {X 0.059,Y -411.207,Z 711.852,A 0.000,B 0.000,C 90.000,E1 189.378} C_DIS
LIN {X 0.151,Y -406.887,Z 711.837,A 0.000,B 0.000,C 90.000,E1 186.606} C_DIS
LIN {X 0.111,Y -404.291,Z 711.827,A 0.000,B 0.000,C 90.000,E1 184.878} C_DIS
LIN {X -0.074,Y -400.925,Z 711.814,A 0.000,B 0.000,C 90.000,E1 182.465} C_DIS
LIN {X -0.098,Y -397.251,Z 711.796,A 0.000,B 0.000,C 90.000,E1 179.312} C_DIS
LIN {X 0.154,Y -394.273,Z 711.779,A 0.000,B 0.000,C 90.000,E1 176.102} C_DIS
LIN {X 0.032,Y -392.139,Z 711.761,A 0.000,B 0.000,C 90.000,E1 172.932} C_DIS
LIN {X 0.090,Y -391.080,Z 711.749,A 0.000,B 0.000,C 90.000,E1 170.792} C_DIS
LIN {X 0.141,Y -390.090,Z 711.733,A 0.000,B 0.000,C 90.000,E1 167.937} C_DIS
LIN {X -0.003,Y -389.304,Z 711.719,A 0.000,B 0.000,C 90.000,E1 165.463} C_DIS
LIN {X 0.068,Y -388.817,Z 711.703,A 0.000,B 0.000,C 90.000,E1 162.598} C_DIS
LIN {X -0.042,Y -388.631,Z 711.690,A 0.000,B 0.000,C 90.000,E1 160.115} C_DIS
LIN {X -0.096,Y -388.558,Z 711.680,A 0.000,B 0.000,C 90.000,E1 158.337} C_DIS
LIN {X 0.018,Y -388.678,Z 711.668,A 0.000,B 0.000,C 90.000,E1 156.177} C_DIS
LIN {X -0.076,Y -388.935,Z 711.654,A 0.000,B 0.000,C 90.000,E1 153.691} C_DIS
LIN {X 0.145,Y -389.131,Z 711.646,A 0.000,B 0.000,C 90.000,E1 152.231} C_DIS
LIN {X -0.001,Y -390.104,Z 711.624,A 0.000,B 0.000,C 90.000,E1 148.329} C_DIS
LIN {X 0.009,Y -392.273,Z 711.604,A 0.000,B 0.000,C 90.000,E1 144.769} C_DIS
LIN {X -0.166,Y -395.635,Z 711.585,A 0.000,B 0.000,C 90.000,E1 141.251} C_DIS
LIN {X 0.024,Y -399.289,Z 711.569,A 0.000,B 0.000,C 90.000,E1 138.405} C_DIS
LIN {X -0.249,Y -400.995,Z 711.563,A 0.000,B 0.000,C 90.000,E1 137.391} C_DIS
LIN {X 0.134,Y -401.754,Z 711.561,A 0.000,B 0.000,C 90.000,E1 136.986} C_DIS
LIN {X 0.098,Y -403.906,Z 711.557,A 0.000,B 0.000,C 90.000,E1 136.296} C_DIS
LIN {X -0.076,Y -405.534,Z 711.555,A 0.000,B 0.000,C 90.000,E1 135.972} C_DIS
LIN {X -0.161,Y -406.462,Z 711.554,A 0.000,B 0.000,C 90.000,E1 135.810} C_DIS
LIN {X 0.172,Y -410.189,Z 711.552,A 0.000,B 0.000,C 90.000,E1 135.243} C_DIS
LIN {X -0.009,Y -414.940,Z 711.548,A 0.000,B 0.000,C 90.000,E1 134.717} C_DIS
LIN {X 0.172,Y -433.695,Z 711.538,A 0.000,B 0.000,C 90.000,E1 132.852} C_DIS
LIN {X -0.146,Y -447.367,Z 711.531,A 0.000,B 0.000,C 90.000,E1 131.676} C_DIS
LIN {X -0.002,Y -460.605,Z 711.525,A 0.000,B 0.000,C 90.000,E1 130.496} C_DIS
LIN {X -0.019,Y -466.498,Z 711.522,A 0.000,B 0.000,C 90.000,E1 129.967} C_DIS
LIN {X -0.179,Y -475.031,Z 711.518,A 0.000,B 0.000,C 90.000,E1 129.197} C_DIS
LIN {X -0.154,Y -480.466,Z 711.515,A 0.000,B 0.000,C 90.000,E1 128.669} C_DIS
LIN {X -0.078,Y -490.245,Z 711.509,A 0.000,B 0.000,C 90.000,E1 127.684} C_DIS
LIN {X 0.076,Y -498.335,Z 711.505,A 0.000,B 0.000,C 90.000,E1 126.824} C_DIS
LIN {X -0.087,Y -506.038,Z 711.500,A 0.000,B 0.000,C 90.000,E1 125.964} C_DIS
LIN {X -0.248,Y -510.951,Z 711.497,A 0.000,B 0.000,C 90.000,E1 125.391} C_DIS
LIN {X 0.110,Y -516.541,Z 711.492,A 0.000,B 0.000,C 90.000,E1 124.612} C_DIS
LIN {X -0.027,Y -520.658,Z 711.489,A 0.000,B 0.000,C 90.000,E1 124.040} C_DIS
LIN {X 0.129,Y -525.199,Z 711.485,A 0.000,B 0.000,C 90.000,E1 123.293} C_DIS
LIN {X -0.113,Y -529.346,Z 711.481,A 0.000,B 0.000,C 90.000,E1 122.594} C_DIS
LIN {X 0.148,Y -531.724,Z 711.479,A 0.000,B 0.000,C 90.000,E1 122.133} C_DIS
LIN {X 0.340,Y -535.981,Z 711.474,A 0.000,B 0.000,C 90.000,E1 121.258} C_DIS
LIN {X -0.095,Y -539.285,Z 711.470,A 0.000,B 0.000,C 90.000,E1 120.590} C_DIS
LIN {X 0.179,Y -544.763,Z 711.463,A 0.000,B 0.000,C 90.000,E1 119.283} C_DIS
LIN {X 0.181,Y -549.315,Z 711.457,A 0.000,B 0.000,C 90.000,E1 118.153} C_DIS
LIN {X -0.043,Y -552.490,Z 711.452,A 0.000,B 0.000,C 90.000,E1 117.334} C_DIS
LIN {X 0.022,Y -555.480,Z 711.447,A 0.000,B 0.000,C 90.000,E1 116.488} C_DIS
LIN {X -0.128,Y -558.228,Z 711.443,A 0.000,B 0.000,C 90.000,E1 115.668} C_DIS
LIN {X -0.012,Y -560.717,Z 711.438,A 0.000,B 0.000,C 90.000,E1 114.823} C_DIS
LIN {X -0.113,Y -562.856,Z 711.433,A 0.000,B 0.000,C 90.000,E1 114.003} C_DIS
LIN {X 0.103,Y -564.797,Z 711.429,A 0.000,B 0.000,C 90.000,E1 113.153} C_DIS
LIN {X 0.048,Y -566.435,Z 711.424,A 0.000,B 0.000,C 90.000,E1 112.333} C_DIS
LIN {X 0.082,Y -569.277,Z 711.415,A 0.000,B 0.000,C 90.000,E1 110.684} C_DIS
LIN {X 0.183,Y -571.949,Z 711.406,A 0.000,B 0.000,C 90.000,E1 109.033} C_DIS
LIN {X -0.023,Y -573.300,Z 711.401,A 0.000,B 0.000,C 90.000,E1 108.236} C_DIS
LIN {X 0.147,Y -575.291,Z 711.394,A 0.000,B 0.000,C 90.000,E1 106.858} C_DIS
LIN {X -0.007,Y -576.892,Z 711.388,A 0.000,B 0.000,C 90.000,E1 105.788} C_DIS
LIN {X 0.077,Y -578.815,Z 711.380,A 0.000,B 0.000,C 90.000,E1 104.426} C_DIS
LIN {X -0.032,Y -580.329,Z 711.374,A 0.000,B 0.000,C 90.000,E1 103.355} C_DIS
LIN {X -0.131,Y -582.965,Z 711.364,A 0.000,B 0.000,C 90.000,E1 101.478} C_DIS
LIN {X 0.051,Y -585.273,Z 711.355,A 0.000,B 0.000,C 90.000,E1 99.849} C_DIS
LIN {X -0.218,Y -586.556,Z 711.349,A 0.000,B 0.000,C 90.000,E1 98.803} C_DIS
LIN {X -0.054,Y -588.456,Z 711.340,A 0.000,B 0.000,C 90.000,E1 97.182} C_DIS
LIN {X 0.077,Y -590.239,Z 711.331,A 0.000,B 0.000,C 90.000,E1 95.568} C_DIS
LIN {X -0.149,Y -592.193,Z 711.321,A 0.000,B 0.000,C 90.000,E1 93.726} C_DIS
LIN {X 0.132,Y -593.144,Z 711.315,A 0.000,B 0.000,C 90.000,E1 92.636} C_DIS
LIN {X -0.168,Y -594.031,Z 711.309,A 0.000,B 0.000,C 90.000,E1 91.604} C_DIS
LIN {X -0.027,Y -595.140,Z 711.300,A 0.000,B 0.000,C 90.000,E1 90.000} C_DIS
LIN {X 0.280,Y -595.620,Z 711.294,A 0.000,B 0.000,C 90.000,E1 88.912} C_DIS
LIN {X 0.238,Y -596.102,Z 711.287,A 0.000,B 0.000,C 90.000,E1 87.593} C_DIS
LIN {X 0.207,Y -596.442,Z 711.279,A 0.000,B 0.000,C 90.000,E1 86.274} C_DIS
LIN {X -0.053,Y -596.649,Z 711.274,A 0.000,B 0.000,C 90.000,E1 85.241} C_DIS
LIN {X 0.019,Y -596.665,Z 711.266,A 0.000,B 0.000,C 90.000,E1 83.913} C_DIS
LIN {X -0.281,Y -596.562,Z 711.257,A 0.000,B 0.000,C 90.000,E1 82.356} C_DIS
LIN {X 0.189,Y -596.358,Z 711.252,A 0.000,B 0.000,C 90.000,E1 81.254} C_DIS
LIN {X 0.253,Y -595.756,Z 711.244,A 0.000,B 0.000,C 90.000,E1 79.926} C_DIS
LIN {X -0.072,Y -594.991,Z 711.237,A 0.000,B 0.000,C 90.000,E1 78.634} C_DIS
LIN {X 0.055,Y -594.041,Z 711.229,A 0.000,B 0.000,C 90.000,E1 77.297} C_DIS
LIN {X -0.156,Y -592.990,Z 711.222,A 0.000,B 0.000,C 90.000,E1 75.992} C_DIS
LIN {X -0.105,Y -591.538,Z 711.213,A 0.000,B 0.000,C 90.000,E1 74.393} C_DIS
LIN {X 0.272,Y -590.765,Z 711.209,A 0.000,B 0.000,C 90.000,E1 73.559} C_DIS
LIN {X -0.134,Y -589.090,Z 711.200,A 0.000,B 0.000,C 90.000,E1 72.000} C_DIS
LIN {X 0.069,Y -587.776,Z 711.194,A 0.000,B 0.000,C 90.000,E1 70.913} C_DIS
LIN {X -0.302,Y -586.475,Z 711.188,A 0.000,B 0.000,C 90.000,E1 69.880} C_DIS
LIN {X -0.068,Y -584.539,Z 711.181,A 0.000,B 0.000,C 90.000,E1 68.518} C_DIS
LIN {X -0.135,Y -583.329,Z 711.176,A 0.000,B 0.000,C 90.000,E1 67.720} C_DIS
LIN {X 0.044,Y -580.969,Z 711.169,A 0.000,B 0.000,C 90.000,E1 66.357} C_DIS
LIN {X 0.023,Y -578.767,Z 711.163,A 0.000,B 0.000,C 90.000,E1 65.281} C_DIS
LIN {X 0.121,Y -576.954,Z 711.158,A 0.000,B 0.000,C 90.000,E1 64.460} C_DIS
LIN {X 0.044,Y -574.289,Z 711.152,A 0.000,B 0.000,C 90.000,E1 63.384} C_DIS
LIN {X 0.084,Y -572.097,Z 711.148,A 0.000,B 0.000,C 90.000,E1 62.564} C_DIS
LIN {X -0.314,Y -568.825,Z 711.142,A 0.000,B 0.000,C 90.000,E1 61.513} C_DIS
LIN {X -0.071,Y -566.223,Z 711.137,A 0.000,B 0.000,C 90.000,E1 60.667} C_DIS
LIN {X -0.349,Y -563.341,Z 711.132,A 0.000,B 0.000,C 90.000,E1 59.871} C_DIS
LIN {X 0.029,Y -561.333,Z 711.129,A 0.000,B 0.000,C 90.000,E1 59.282} C_DIS
LIN {X -0.010,Y -557.951,Z 711.125,A 0.000,B 0.000,C 90.000,E1 58.456} C_DIS
LIN {X -0.263,Y -554.901,Z 711.121,A 0.000,B 0.000,C 90.000,E1 57.788} C_DIS
LIN {X 0.219,Y -551.429,Z 711.117,A 0.000,B 0.000,C 90.000,E1 57.041} C_DIS
LIN {X 0.076,Y -546.674,Z 711.112,A 0.000,B 0.000,C 90.000,E1 56.215} C_DIS
LIN {X -0.148,Y -543.255,Z 711.109,A 0.000,B 0.000,C 90.000,E1 55.674} C_DIS
LIN {X -0.089,Y -539.624,Z 711.106,A 0.000,B 0.000,C 90.000,E1 55.102} C_DIS
LIN {X -0.053,Y -535.653,Z 711.103,A 0.000,B 0.000,C 90.000,E1 54.529} C_DIS
LIN {X -0.356,Y -531.187,Z 711.100,A 0.000,B 0.000,C 90.000,E1 53.989} C_DIS
LIN {X 0.044,Y -526.219,Z 711.097,A 0.000,B 0.000,C 90.000,E1 53.371} C_DIS
LIN {X 0.242,Y -522.275,Z 711.094,A 0.000,B 0.000,C 90.000,E1 52.924} C_DIS
LIN {X -0.083,Y -518.030,Z 711.092,A 0.000,B 0.000,C 90.000,E1 52.557} C_DIS
LIN {X 0.094,Y -512.540,Z 711.089,A 0.000,B 0.000,C 90.000,E1 52.065} C_DIS
LIN {X -0.159,Y -505.321,Z 711.086,A 0.000,B 0.000,C 90.000,E1 51.537} C_DIS
LIN {X 0.075,Y -497.252,Z 711.083,A 0.000,B 0.000,C 90.000,E1 50.964} C_DIS
LIN {X 0.156,Y -489.102,Z 711.080,A 0.000,B 0.000,C 90.000,E1 50.436} C_DIS
LIN {X 0.216,Y -472.777,Z 711.075,A 0.000,B 0.000,C 90.000,E1 49.461} C_DIS
LIN {X -0.054,Y -453.439,Z 711.068,A 0.000,B 0.000,C 90.000,E1 48.324} C_DIS
LIN {X 0.126,Y -434.194,Z 711.062,A 0.000,B 0.000,C 90.000,E1 47.067} C_DIS
LIN {X 0.227,Y -423.486,Z 711.057,A 0.000,B 0.000,C 90.000,E1 46.296} C_DIS
LIN {X 0.036,Y -421.040,Z 711.056,A 0.000,B 0.000,C 90.000,E1 46.134} C_DIS
LIN {X 0.009,Y -421.005,Z 711.056,A 0.000,B 0.000,C 90.000,E1 46.134} C_DIS
LIN {X -0.189,Y -418.432,Z 711.049,A 0.000,B 0.000,C 90.000,E1 44.757} C_DIS
LIN {X -0.101,Y -408.901,Z 711.024,A 0.000,B 0.000,C 90.000,E1 40.297} C_DIS
LIN {X 0.053,Y -408.284,Z 711.022,A 0.000,B 0.000,C 90.000,E1 39.930} C_DIS
LIN {X 0.206,Y -408.170,Z 711.020,A 0.000,B 0.000,C 90.000,E1 39.564} C_DIS
LIN {X 0.114,Y -408.385,Z 711.007,A 0.000,B 0.000,C 90.000,E1 37.156} C_DIS
LIN {X -0.060,Y -409.400,Z 710.989,A 0.000,B 0.000,C 90.000,E1 34.072} C_DIS
LIN {X -0.160,Y -410.493,Z 710.976,A 0.000,B 0.000,C 90.000,E1 31.671} C_DIS
LIN {X 0.036,Y -411.354,Z 710.966,A 0.000,B 0.000,C 90.000,E1 29.922} C_DIS
LIN {X -0.163,Y -412.339,Z 710.957,A 0.000,B 0.000,C 90.000,E1 28.231} C_DIS
LIN {X 0.001,Y -414.097,Z 710.942,A 0.000,B 0.000,C 90.000,E1 25.463} C_DIS
LIN {X 0.171,Y -415.684,Z 710.930,A 0.000,B 0.000,C 90.000,E1 23.387} C_DIS
LIN {X 0.129,Y -418.156,Z 710.915,A 0.000,B 0.000,C 90.000,E1 20.663} C_DIS
LIN {X -0.078,Y -420.274,Z 710.904,A 0.000,B 0.000,C 90.000,E1 18.652} C_DIS
LIN {X 0.252,Y -422.200,Z 710.894,A 0.000,B 0.000,C 90.000,E1 16.913} C_DIS
LIN {X -0.054,Y -425.103,Z 710.881,A 0.000,B 0.000,C 90.000,E1 14.592} C_DIS
LIN {X -0.170,Y -427.736,Z 710.870,A 0.000,B 0.000,C 90.000,E1 12.591} C_DIS
LIN {X 0.002,Y -430.000,Z 710.861,A 0.000,B 0.000,C 90.000,E1 10.894} C_DIS
LIN {X -0.169,Y -432.730,Z 710.849,A 0.000,B 0.000,C 90.000,E1 8.916} C_DIS
LIN {X 0.083,Y -435.559,Z 710.838,A 0.000,B 0.000,C 90.000,E1 6.891} C_DIS
LIN {X -0.128,Y -438.422,Z 710.827,A 0.000,B 0.000,C 90.000,E1 4.935} C_DIS
LIN {X -0.039,Y -442.576,Z 710.813,A 0.000,B 0.000,C 90.000,E1 2.293} C_DIS
LIN {X 0.169,Y -446.944,Z 710.799,A 0.000,B 0.000,C 90.000,E1 359.771} C_DIS
LIN {X 0.025,Y -450.039,Z 710.790,A 0.000,B 0.000,C 90.000,E1 358.165} C_DIS
LIN {X 0.019,Y -455.138,Z 710.776,A 0.000,B 0.000,C 90.000,E1 355.584} C_DIS
LIN {X -0.180,Y -459.093,Z 710.765,A 0.000,B 0.000,C 90.000,E1 353.685} C_DIS
LIN {X 0.032,Y -462.395,Z 710.756,A 0.000,B 0.000,C 90.000,E1 352.064} C_DIS
LIN {X -0.079,Y -466.761,Z 710.744,A 0.000,B 0.000,C 90.000,E1 349.859} C_DIS
LIN {X 0.085,Y -469.178,Z 710.737,A 0.000,B 0.000,C 90.000,E1 348.578} C_DIS
LIN {X 0.206,Y -471.995,Z 710.728,A 0.000,B 0.000,C 90.000,E1 346.992} C_DIS
LIN {X 0.163,Y -476.075,Z 710.716,A 0.000,B 0.000,C 90.000,E1 344.810} C_DIS
LIN {X -0.122,Y -480.132,Z 710.704,A 0.000,B 0.000,C 90.000,E1 342.670} C_DIS
LIN {X -0.021,Y -484.540,Z 710.692,A 0.000,B 0.000,C 90.000,E1 340.496} C_DIS
LIN {X 0.037,Y -487.904,Z 710.683,A 0.000,B 0.000,C 90.000,E1 338.954} C_DIS
LIN {X 0.083,Y -489.547,Z 710.680,A 0.000,B 0.000,C 90.000,E1 338.337} C_DIS
LIN {X 0.155,Y -491.705,Z 710.676,A 0.000,B 0.000,C 90.000,E1 337.720} C_DIS
LIN {X 0.225,Y -493.185,Z 710.675,A 0.000,B 0.000,C 90.000,E1 337.411} C_DIS
LIN {X 0.071,Y -495.388,Z 710.673,A 0.000,B 0.000,C 90.000,E1 337.102} C_DIS
LIN {X -0.099,Y -498.229,Z 710.671,A 0.000,B 0.000,C 90.000,E1 336.794} C_DIS
LIN {X 0.071,Y -501.040,Z 710.669,A 0.000,B 0.000,C 90.000,E1 336.485} C_DIS
LIN {X -0.187,Y -504.824,Z 710.668,A 0.000,B 0.000,C 90.000,E1 336.177} C_DIS
LIN {X -0.182,Y -515.698,Z 710.663,A 0.000,B 0.000,C 90.000,E1 335.409} C_DIS
LIN {X 0.218,Y -531.526,Z 710.658,A 0.000,B 0.000,C 90.000,E1 334.332} C_DIS
LIN {X 0.004,Y -539.159,Z 710.655,A 0.000,B 0.000,C 90.000,E1 333.819} C_DIS
LIN {X -0.056,Y -545.145,Z 710.652,A 0.000,B 0.000,C 90.000,E1 333.384} C_DIS
LIN {X 0.110,Y -553.693,Z 710.648,A 0.000,B 0.000,C 90.000,E1 332.666} C_DIS
LIN {X 0.111,Y -559.038,Z 710.646,A 0.000,B 0.000,C 90.000,E1 332.180} C_DIS
LIN {X -0.086,Y -564.394,Z 710.643,A 0.000,B 0.000,C 90.000,E1 331.691} C_DIS
LIN {X -0.154,Y -570.753,Z 710.639,A 0.000,B 0.000,C 90.000,E1 331.051} C_DIS
LIN {X 0.172,Y -579.502,Z 710.634,A 0.000,B 0.000,C 90.000,E1 330.078} C_DIS
LIN {X 0.070,Y -586.632,Z 710.629,A 0.000,B 0.000,C 90.000,E1 329.282} C_DIS
LIN {X 0.007,Y -593.486,Z 710.625,A 0.000,B 0.000,C 90.000,E1 328.486} C_DIS
LIN {X 0.107,Y -598.007,Z 710.622,A 0.000,B 0.000,C 90.000,E1 327.946} C_DIS
LIN {X -0.026,Y -604.403,Z 710.618,A 0.000,B 0.000,C 90.000,E1 327.168} C_DIS
LIN {X 0.088,Y -610.365,Z 710.613,A 0.000,B 0.000,C 90.000,E1 326.373} C_DIS
LIN {X 0.090,Y -616.012,Z 710.609,A 0.000,B 0.000,C 90.000,E1 325.595} C_DIS
LIN {X -0.160,Y -619.578,Z 710.606,A 0.000,B 0.000,C 90.000,E1 325.102} C_DIS
LIN {X 0.005,Y -625.417,Z 710.601,A 0.000,B 0.000,C 90.000,E1 324.196} C_DIS
LIN {X 0.158,Y -630.946,Z 710.596,A 0.000,B 0.000,C 90.000,E1 323.290} C_DIS
LIN {X 0.247,Y -636.815,Z 710.591,A 0.000,B 0.000,C 90.000,E1 322.271} C_DIS
LIN {X -0.079,Y -643.730,Z 710.584,A 0.000,B 0.000,C 90.000,E1 321.045} C_DIS
LIN {X 0.098,Y -649.627,Z 710.577,A 0.000,B 0.000,C 90.000,E1 319.908} C_DIS
LIN {X -0.064,Y -654.547,Z 710.572,A 0.000,B 0.000,C 90.000,E1 318.933} C_DIS
LIN {X 0.266,Y -659.190,Z 710.566,A 0.000,B 0.000,C 90.000,E1 317.919} C_DIS
LIN {X -0.257,Y -662.425,Z 710.562,A 0.000,B 0.000,C 90.000,E1 317.229} C_DIS
LIN {X 0.178,Y -666.530,Z 710.557,A 0.000,B 0.000,C 90.000,E1 316.215} C_DIS
LIN {X 0.180,Y -669.297,Z 710.553,A 0.000,B 0.000,C 90.000,E1 315.486} C_DIS
LIN {X 0.266,Y -674.553,Z 710.545,A 0.000,B 0.000,C 90.000,E1 314.028} C_DIS
LIN {X -0.055,Y -678.577,Z 710.538,A 0.000,B 0.000,C 90.000,E1 312.852} C_DIS
LIN {X -0.317,Y -682.431,Z 710.531,A 0.000,B 0.000,C 90.000,E1 311.676} C_DIS
LIN {X -0.013,Y -685.901,Z 710.525,A 0.000,B 0.000,C 90.000,E1 310.458} C_DIS
LIN {X 0.230,Y -687.832,Z 710.521,A 0.000,B 0.000,C 90.000,E1 309.725} C_DIS
LIN {X -0.415,Y -690.017,Z 710.516,A 0.000,B 0.000,C 90.000,E1 308.830} C_DIS
LIN {X -0.127,Y -691.544,Z 710.512,A 0.000,B 0.000,C 90.000,E1 308.096} C_DIS
LIN {X -0.189,Y -693.272,Z 710.506,A 0.000,B 0.000,C 90.000,E1 307.156} C_DIS
LIN {X -0.021,Y -695.167,Z 710.500,A 0.000,B 0.000,C 90.000,E1 305.964} C_DIS
LIN {X -0.042,Y -696.452,Z 710.495,A 0.000,B 0.000,C 90.000,E1 305.025} C_DIS
LIN {X 0.171,Y -697.819,Z 710.488,A 0.000,B 0.000,C 90.000,E1 303.833} C_DIS
LIN {X -0.272,Y -698.533,Z 710.484,A 0.000,B 0.000,C 90.000,E1 303.166} C_DIS
LIN {X -0.129,Y -699.961,Z 710.475,A 0.000,B 0.000,C 90.000,E1 301.514} C_DIS
LIN {X -0.285,Y -700.656,Z 710.470,A 0.000,B 0.000,C 90.000,E1 300.590} C_DIS
LIN {X 0.181,Y -701.047,Z 710.465,A 0.000,B 0.000,C 90.000,E1 299.617} C_DIS
LIN {X 0.256,Y -701.544,Z 710.456,A 0.000,B 0.000,C 90.000,E1 297.975} C_DIS
LIN {X -0.094,Y -702.580,Z 710.443,A 0.000,B 0.000,C 90.000,E1 295.668} C_DIS
LIN {X -0.169,Y -702.725,Z 710.440,A 0.000,B 0.000,C 90.000,E1 295.207} C_DIS
LIN {X 0.094,Y -702.267,Z 710.437,A 0.000,B 0.000,C 90.000,E1 294.719} C_DIS
LIN {X -0.265,Y -701.949,Z 710.436,A 0.000,B 0.000,C 90.000,E1 294.515} C_DIS
LIN {X 0.011,Y -701.051,Z 710.435,A 0.000,B 0.000,C 90.000,E1 294.259} C_DIS
LIN {X 0.135,Y -699.253,Z 710.433,A 0.000,B 0.000,C 90.000,E1 293.898} C_DIS
LIN {X 0.271,Y -698.575,Z 710.432,A 0.000,B 0.000,C 90.000,E1 293.770} C_DIS
LIN {X -0.236,Y -697.600,Z 710.432,A 0.000,B 0.000,C 90.000,E1 293.695} C_DIS
LIN {X -0.105,Y -696.141,Z 710.431,A 0.000,B 0.000,C 90.000,E1 293.567} C_DIS
LIN {X -0.052,Y -691.157,Z 710.429,A 0.000,B 0.000,C 90.000,E1 293.259} C_DIS
LIN {X 0.106,Y -689.515,Z 710.429,A 0.000,B 0.000,C 90.000,E1 293.153} C_DIS
LIN {X -0.021,Y -687.344,Z 710.428,A 0.000,B 0.000,C 90.000,E1 293.078} C_DIS
LIN {X -0.147,Y -683.998,Z 710.428,A 0.000,B 0.000,C 90.000,E1 293.003} C_DIS
LIN {X 0.194,Y -677.998,Z 710.427,A 0.000,B 0.000,C 90.000,E1 292.845} C_DIS
LIN {X -0.097,Y -660.230,Z 710.426,A 0.000,B 0.000,C 90.000,E1 292.642} C_DIS
LIN {X 0.119,Y -646.364,Z 710.425,A 0.000,B 0.000,C 90.000,E1 292.408} C_DIS
LIN {X 0.306,Y -636.627,Z 710.424,A 0.000,B 0.000,C 90.000,E1 292.206} C_DIS
LIN {X 0.338,Y -623.305,Z 710.422,A 0.000,B 0.000,C 90.000,E1 291.897} C_DIS
LIN {X 0.092,Y -606.145,Z 710.419,A 0.000,B 0.000,C 90.000,E1 291.461} C_DIS
LIN {X -0.173,Y -578.374,Z 710.415,A 0.000,B 0.000,C 90.000,E1 290.663} C_DIS
LIN {X -0.157,Y -568.121,Z 710.413,A 0.000,B 0.000,C 90.000,E1 290.355} C_DIS
LIN {X 0.050,Y -562.081,Z 710.412,A 0.000,B 0.000,C 90.000,E1 290.120} C_DIS
LIN {X 0.228,Y -559.631,Z 710.411,A 0.000,B 0.000,C 90.000,E1 289.993} C_DIS
LIN {X 0.114,Y -556.052,Z 710.410,A 0.000,B 0.000,C 90.000,E1 289.758} C_DIS
LIN {X 0.082,Y -556.020,Z 710.410,A 0.000,B 0.000,C 90.000,E1 289.758} C_DIS
LIN {X -0.227,Y -555.320,Z 710.409,A 0.000,B 0.000,C 90.000,E1 289.631} C_DIS
LIN {X -0.209,Y -554.710,Z 710.406,A 0.000,B 0.000,C 90.000,E1 289.141} C_DIS
LIN {X 0.318,Y -554.126,Z 710.398,A 0.000,B 0.000,C 90.000,E1 287.692} C_DIS
LIN {X 0.252,Y -553.473,Z 710.389,A 0.000,B 0.000,C 90.000,E1 286.024} C_DIS
LIN {X -0.245,Y -552.788,Z 710.378,A 0.000,B 0.000,C 90.000,E1 284.120} C_DIS
LIN {X -0.064,Y -552.300,Z 710.371,A 0.000,B 0.000,C 90.000,E1 282.703} C_DIS
LIN {X -0.017,Y -551.744,Z 710.363,A 0.000,B 0.000,C 90.000,E1 281.299} C_DIS
LIN {X -0.079,Y -551.094,Z 710.355,A 0.000,B 0.000,C 90.000,E1 279.905} C_DIS
LIN {X -0.009,Y -550.228,Z 710.344,A 0.000,B 0.000,C 90.000,E1 277.936} C_DIS
LIN {X -0.068,Y -549.584,Z 710.335,A 0.000,B 0.000,C 90.000,E1 276.258} C_DIS
LIN {X -0.078,Y -549.086,Z 710.322,A 0.000,B 0.000,C 90.000,E1 274.012} C_DIS
LIN {X 0.142,Y -548.754,Z 710.316,A 0.000,B 0.000,C 90.000,E1 272.865} C_DIS
LIN {X -0.095,Y -548.193,Z 710.307,A 0.000,B 0.000,C 90.000,E1 271.203} C_DIS
LIN {X 0.100,Y -547.643,Z 710.300,A 0.000,B 0.000,C 90.000,E1 270.057} C_DIS
LIN {X -0.112,Y -546.416,Z 710.289,A 0.000,B 0.000,C 90.000,E1 268.108} C_DIS
LIN {X 0.115,Y -545.607,Z 710.282,A 0.000,B 0.000,C 90.000,E1 266.674} C_DIS
LIN {X -0.227,Y -544.570,Z 710.274,A 0.000,B 0.000,C 90.000,E1 265.298} C_DIS
LIN {X 0.060,Y -543.330,Z 710.264,A 0.000,B 0.000,C 90.000,E1 263.571} C_DIS
LIN {X -0.236,Y -542.349,Z 710.258,A 0.000,B 0.000,C 90.000,E1 262.470} C_DIS
LIN {X 0.070,Y -540.832,Z 710.249,A 0.000,B 0.000,C 90.000,E1 260.735} C_DIS
LIN {X -0.186,Y -539.546,Z 710.241,A 0.000,B 0.000,C 90.000,E1 259.342} C_DIS
LIN {X -0.232,Y -537.757,Z 710.230,A 0.000,B 0.000,C 90.000,E1 257.353} C_DIS
LIN {X -0.077,Y -535.880,Z 710.219,A 0.000,B 0.000,C 90.000,E1 255.338} C_DIS
LIN {X 0.269,Y -534.770,Z 710.212,A 0.000,B 0.000,C 90.000,E1 254.157} C_DIS
LIN {X -0.210,Y -533.038,Z 710.203,A 0.000,B 0.000,C 90.000,E1 252.489} C_DIS
LIN {X -0.089,Y -531.582,Z 710.195,A 0.000,B 0.000,C 90.000,E1 251.040} C_DIS
LIN {X -0.006,Y -530.211,Z 710.188,A 0.000,B 0.000,C 90.000,E1 249.880} C_DIS
LIN {X 0.240,Y -528.283,Z 710.180,A 0.000,B 0.000,C 90.000,E1 248.411} C_DIS
LIN {X -0.017,Y -526.634,Z 710.174,A 0.000,B 0.000,C 90.000,E1 247.283} C_DIS
LIN {X 0.192,Y -524.955,Z 710.167,A 0.000,B 0.000,C 90.000,E1 246.102} C_DIS
LIN {X -0.270,Y -522.070,Z 710.158,A 0.000,B 0.000,C 90.000,E1 244.409} C_DIS
LIN {X 0.076,Y -520.054,Z 710.151,A 0.000,B 0.000,C 90.000,E1 243.204} C_DIS
LIN {X -0.169,Y -517.198,Z 710.143,A 0.000,B 0.000,C 90.000,E1 241.769} C_DIS
LIN {X -0.116,Y -514.909,Z 710.137,A 0.000,B 0.000,C 90.000,E1 240.589} C_DIS
LIN {X -0.192,Y -511.805,Z 710.128,A 0.000,B 0.000,C 90.000,E1 239.125} C_DIS
LIN {X 0.004,Y -508.027,Z 710.119,A 0.000,B 0.000,C 90.000,E1 237.327} C_DIS
LIN {X 0.340,Y -504.902,Z 710.110,A 0.000,B 0.000,C 90.000,E1 235.801} C_DIS
LIN {X 0.029,Y -502.276,Z 710.104,A 0.000,B 0.000,C 90.000,E1 234.642} C_DIS
LIN {X 0.092,Y -500.942,Z 710.100,A 0.000,B 0.000,C 90.000,E1 234.036} C_DIS
LIN {X 0.012,Y -497.907,Z 710.094,A 0.000,B 0.000,C 90.000,E1 232.844} C_DIS
LIN {X 0.062,Y -492.523,Z 710.082,A 0.000,B 0.000,C 90.000,E1 230.723} C_DIS
LIN {X -0.090,Y -487.454,Z 710.070,A 0.000,B 0.000,C 90.000,E1 228.609} C_DIS
LIN {X 0.139,Y -483.241,Z 710.060,A 0.000,B 0.000,C 90.000,E1 226.743} C_DIS
LIN {X 0.007,Y -480.511,Z 710.053,A 0.000,B 0.000,C 90.000,E1 225.526} C_DIS
LIN {X 0.061,Y -476.436,Z 710.043,A 0.000,B 0.000,C 90.000,E1 223.662} C_DIS
LIN {X 0.134,Y -471.688,Z 710.031,A 0.000,B 0.000,C 90.000,E1 221.472} C_DIS
LIN {X -0.080,Y -468.327,Z 710.022,A 0.000,B 0.000,C 90.000,E1 219.930} C_DIS
LIN {X -0.064,Y -465.660,Z 710.015,A 0.000,B 0.000,C 90.000,E1 218.669} C_DIS
LIN {X -0.088,Y -460.133,Z 710.001,A 0.000,B 0.000,C 90.000,E1 216.137} C_DIS
LIN {X 0.258,Y -457.527,Z 709.994,A 0.000,B 0.000,C 90.000,E1 214.818} C_DIS
LIN {X -0.172,Y -455.741,Z 709.988,A 0.000,B 0.000,C 90.000,E1 213.913} C_DIS
LIN {X 0.054,Y -452.093,Z 709.978,A 0.000,B 0.000,C 90.000,E1 211.957} C_DIS
LIN {X -0.264,Y -447.288,Z 709.963,A 0.000,B 0.000,C 90.000,E1 209.411} C_DIS
LIN {X -0.236,Y -443.183,Z 709.951,A 0.000,B 0.000,C 90.000,E1 207.129} C_DIS
LIN {X -0.168,Y -439.606,Z 709.940,A 0.000,B 0.000,C 90.000,E1 205.155} C_DIS
LIN {X 0.032,Y -435.949,Z 709.929,A 0.000,B 0.000,C 90.000,E1 203.153} C_DIS
LIN {X -0.075,Y -433.518,Z 709.921,A 0.000,B 0.000,C 90.000,E1 201.844} C_DIS
LIN {X 0.207,Y -429.903,Z 709.910,A 0.000,B 0.000,C 90.000,E1 199.812} C_DIS
LIN {X -0.095,Y -426.859,Z 709.901,A 0.000,B 0.000,C 90.000,E1 198.181} C_DIS
LIN {X 0.136,Y -423.199,Z 709.890,A 0.000,B 0.000,C 90.000,E1 196.134} C_DIS
LIN {X 0.039,Y -419.480,Z 709.879,A 0.000,B 0.000,C 90.000,E1 194.120} C_DIS
LIN {X -0.142,Y -414.712,Z 709.863,A 0.000,B 0.000,C 90.000,E1 191.422} C_DIS
LIN {X 0.188,Y -411.195,Z 709.852,A 0.000,B 0.000,C 90.000,E1 189.321} C_DIS
LIN {X -0.122,Y -406.899,Z 709.837,A 0.000,B 0.000,C 90.000,E1 186.606} C_DIS
LIN {X -0.161,Y -404.302,Z 709.827,A 0.000,B 0.000,C 90.000,E1 184.878} C_DIS
LIN {X 0.056,Y -400.942,Z 709.813,A 0.000,B 0.000,C 90.000,E1 182.407} C_DIS
LIN {X 0.088,Y -397.695,Z 709.798,A 0.000,B 0.000,C 90.000,E1 179.599} C_DIS
LIN {X -0.107,Y -394.343,Z 709.778,A 0.000,B 0.000,C 90.000,E1 176.102} C_DIS
LIN {X 0.068,Y -392.079,Z 709.759,A 0.000,B 0.000,C 90.000,E1 172.534} C_DIS
LIN {X 0.175,Y -391.071,Z 709.747,A 0.000,B 0.000,C 90.000,E1 170.387} C_DIS
LIN {X -0.107,Y -390.266,Z 709.733,A 0.000,B 0.000,C 90.000,E1 167.937} C_DIS
LIN {X 0.194,Y -389.595,Z 709.721,A 0.000,B 0.000,C 90.000,E1 165.755} C_DIS
LIN {X -0.167,Y -389.017,Z 709.703,A 0.000,B 0.000,C 90.000,E1 162.598} C_DIS
LIN {X 0.094,Y -388.845,Z 709.689,A 0.000,B 0.000,C 90.000,E1 160.061} C_DIS
LIN {X 0.072,Y -388.784,Z 709.677,A 0.000,B 0.000,C 90.000,E1 157.922} C_DIS
LIN {X -0.202,Y -388.921,Z 709.668,A 0.000,B 0.000,C 90.000,E1 156.177} C_DIS
LIN {X 0.060,Y -389.210,Z 709.654,A 0.000,B 0.000,C 90.000,E1 153.640} C_DIS
LIN {X -0.062,Y -389.370,Z 709.646,A 0.000,B 0.000,C 90.000,E1 152.231} C_DIS
LIN {X -0.046,Y -390.238,Z 709.626,A 0.000,B 0.000,C 90.000,E1 148.663} C_DIS
LIN {X -0.102,Y -391.966,Z 709.608,A 0.000,B 0.000,C 90.000,E1 145.468} C_DIS
LIN {X -0.003,Y -393.969,Z 709.594,A 0.000,B 0.000,C 90.000,E1 142.970} C_DIS
LIN {X -0.165,Y -397.890,Z 709.575,A 0.000,B 0.000,C 90.000,E1 139.461} C_DIS
LIN {X 0.137,Y -400.918,Z 709.563,A 0.000,B 0.000,C 90.000,E1 137.310} C_DIS
LIN {X -0.047,Y -401.605,Z 709.561,A 0.000,B 0.000,C 90.000,E1 136.986} C_DIS
LIN {X 0.064,Y -402.688,Z 709.559,A 0.000,B 0.000,C 90.000,E1 136.620} C_DIS
LIN {X -0.115,Y -403.602,Z 709.557,A 0.000,B 0.000,C 90.000,E1 136.296} C_DIS
LIN {X 0.197,Y -405.919,Z 709.554,A 0.000,B 0.000,C 90.000,E1 135.729} C_DIS
LIN {X 0.113,Y -406.796,Z 709.553,A 0.000,B 0.000,C 90.000,E1 135.567} C_DIS
LIN {X -0.061,Y -409.139,Z 709.551,A 0.000,B 0.000,C 90.000,E1 135.243} C_DIS
LIN {X -0.216,Y -414.073,Z 709.548,A 0.000,B 0.000,C 90.000,E1 134.676} C_DIS
LIN {X -0.183,Y -435.174,Z 709.537,A 0.000,B 0.000,C 90.000,E1 132.609} C_DIS
LIN {X 0.059,Y -445.846,Z 709.531,A 0.000,B 0.000,C 90.000,E1 131.634} C_DIS
LIN {X -0.300,Y -458.096,Z 709.526,A 0.000,B 0.000,C 90.000,E1 130.620} C_DIS
LIN {X -0.032,Y -465.483,Z 709.522,A 0.000,B 0.000,C 90.000,E1 129.930} C_DIS
LIN {X 0.057,Y -474.284,Z 709.517,A 0.000,B 0.000,C 90.000,E1 129.116} C_DIS
LIN {X -0.089,Y -479.941,Z 709.514,A 0.000,B 0.000,C 90.000,E1 128.588} C_DIS
LIN {X 0.054,Y -489.747,Z 709.509,A 0.000,B 0.000,C 90.000,E1 127.604} C_DIS
LIN {X 0.137,Y -497.932,Z 709.504,A 0.000,B 0.000,C 90.000,E1 126.744} C_DIS
LIN {X 0.027,Y -505.711,Z 709.499,A 0.000,B 0.000,C 90.000,E1 125.884} C_DIS
LIN {X 0.064,Y -509.429,Z 709.497,A 0.000,B 0.000,C 90.000,E1 125.438} C_DIS
LIN {X 0.059,Y -511.795,Z 709.495,A 0.000,B 0.000,C 90.000,E1 125.152} C_DIS
LIN {X 0.046,Y -517.034,Z 709.491,A 0.000,B 0.000,C 90.000,E1 124.452} C_DIS
LIN {X 0.225,Y -520.186,Z 709.489,A 0.000,B 0.000,C 90.000,E1 123.992} C_DIS
LIN {X 0.202,Y -524.688,Z 709.485,A 0.000,B 0.000,C 90.000,E1 123.293} C_DIS
LIN {X -0.002,Y -528.095,Z 709.482,A 0.000,B 0.000,C 90.000,E1 122.752} C_DIS
LIN {X 0.226,Y -532.095,Z 709.478,A 0.000,B 0.000,C 90.000,E1 122.005} C_DIS
LIN {X -0.242,Y -535.733,Z 709.474,A 0.000,B 0.000,C 90.000,E1 121.337} C_DIS
LIN {X 0.058,Y -539.107,Z 709.470,A 0.000,B 0.000,C 90.000,E1 120.590} C_DIS
LIN {X -0.143,Y -544.633,Z 709.463,A 0.000,B 0.000,C 90.000,E1 119.333} C_DIS
LIN {X 0.075,Y -549.205,Z 709.457,A 0.000,B 0.000,C 90.000,E1 118.180} C_DIS
LIN {X 0.110,Y -552.414,Z 709.452,A 0.000,B 0.000,C 90.000,E1 117.334} C_DIS
LIN {X 0.175,Y -555.433,Z 709.447,A 0.000,B 0.000,C 90.000,E1 116.488} C_DIS
LIN {X 0.024,Y -558.245,Z 709.443,A 0.000,B 0.000,C 90.000,E1 115.668} C_DIS
LIN {X 0.142,Y -560.765,Z 709.438,A 0.000,B 0.000,C 90.000,E1 114.823} C_DIS
LIN {X -0.186,Y -562.942,Z 709.433,A 0.000,B 0.000,C 90.000,E1 114.027} C_DIS
LIN {X -0.259,Y -564.949,Z 709.429,A 0.000,B 0.000,C 90.000,E1 113.206} C_DIS
LIN {X 0.206,Y -566.624,Z 709.424,A 0.000,B 0.000,C 90.000,E1 112.333} C_DIS
LIN {X -0.287,Y -569.497,Z 709.415,A 0.000,B 0.000,C 90.000,E1 110.737} C_DIS
LIN {X -0.188,Y -572.170,Z 709.406,A 0.000,B 0.000,C 90.000,E1 109.087} C_DIS
LIN {X -0.218,Y -573.967,Z 709.400,A 0.000,B 0.000,C 90.000,E1 108.000} C_DIS
LIN {X -0.033,Y -575.988,Z 709.392,A 0.000,B 0.000,C 90.000,E1 106.622} C_DIS
LIN {X 0.185,Y -577.975,Z 709.385,A 0.000,B 0.000,C 90.000,E1 105.245} C_DIS
LIN {X -0.061,Y -580.323,Z 709.376,A 0.000,B 0.000,C 90.000,E1 103.647} C_DIS
LIN {X 0.072,Y -583.360,Z 709.364,A 0.000,B 0.000,C 90.000,E1 101.478} C_DIS
LIN {X 0.263,Y -585.696,Z 709.355,A 0.000,B 0.000,C 90.000,E1 99.849} C_DIS
LIN {X 0.000,Y -586.997,Z 709.349,A 0.000,B 0.000,C 90.000,E1 98.803} C_DIS
LIN {X 0.175,Y -588.929,Z 709.340,A 0.000,B 0.000,C 90.000,E1 97.182} C_DIS
LIN {X -0.126,Y -590.079,Z 709.334,A 0.000,B 0.000,C 90.000,E1 96.144} C_DIS
LIN {X 0.175,Y -591.281,Z 709.328,A 0.000,B 0.000,C 90.000,E1 95.049} C_DIS
LIN {X 0.102,Y -592.717,Z 709.321,A 0.000,B 0.000,C 90.000,E1 93.726} C_DIS
LIN {X -0.201,Y -593.676,Z 709.315,A 0.000,B 0.000,C 90.000,E1 92.694} C_DIS
LIN {X 0.098,Y -594.577,Z 709.309,A 0.000,B 0.000,C 90.000,E1 91.604} C_DIS
LIN {X 0.252,Y -595.707,Z 709.300,A 0.000,B 0.000,C 90.000,E1 90.000} C_DIS
LIN {X -0.258,Y -596.085,Z 709.296,A 0.000,B 0.000,C 90.000,E1 89.255} C_DIS
LIN {X -0.060,Y -596.661,Z 709.287,A 0.000,B 0.000,C 90.000,E1 87.650} C_DIS
LIN {X -0.082,Y -597.003,Z 709.280,A 0.000,B 0.000,C 90.000,E1 86.331} C_DIS
LIN {X -0.059,Y -597.235,Z 709.272,A 0.000,B 0.000,C 90.000,E1 85.008} C_DIS
LIN {X -0.033,Y -597.220,Z 709.265,A 0.000,B 0.000,C 90.000,E1 83.685} C_DIS
LIN {X -0.331,Y -597.070,Z 709.256,A 0.000,B 0.000,C 90.000,E1 82.129} C_DIS
LIN {X 0.140,Y -596.783,Z 709.250,A 0.000,B 0.000,C 90.000,E1 81.027} C_DIS
LIN {X -0.280,Y -596.115,Z 709.243,A 0.000,B 0.000,C 90.000,E1 79.746} C_DIS
LIN {X 0.289,Y -595.500,Z 709.237,A 0.000,B 0.000,C 90.000,E1 78.634} C_DIS
LIN {X -0.157,Y -594.521,Z 709.230,A 0.000,B 0.000,C 90.000,E1 77.353} C_DIS
LIN {X 0.220,Y -593.431,Z 709.222,A 0.000,B 0.000,C 90.000,E1 75.992} C_DIS
LIN {X 0.012,Y -592.178,Z 709.215,A 0.000,B 0.000,C 90.000,E1 74.685} C_DIS
LIN {X 0.092,Y -591.182,Z 709.209,A 0.000,B 0.000,C 90.000,E1 73.614} C_DIS
LIN {X 0.260,Y -589.444,Z 709.200,A 0.000,B 0.000,C 90.000,E1 72.000} C_DIS
LIN {X -0.088,Y -588.139,Z 709.194,A 0.000,B 0.000,C 90.000,E1 70.967} C_DIS
LIN {X 0.100,Y -586.776,Z 709.188,A 0.000,B 0.000,C 90.000,E1 69.880} C_DIS
LIN {X -0.008,Y -584.385,Z 709.179,A 0.000,B 0.000,C 90.000,E1 68.284} C_DIS
LIN {X 0.051,Y -583.580,Z 709.176,A 0.000,B 0.000,C 90.000,E1 67.741} C_DIS
LIN {X -0.079,Y -581.144,Z 709.169,A 0.000,B 0.000,C 90.000,E1 66.410} C_DIS
LIN {X -0.334,Y -578.927,Z 709.163,A 0.000,B 0.000,C 90.000,E1 65.357} C_DIS
LIN {X -0.237,Y -577.075,Z 709.158,A 0.000,B 0.000,C 90.000,E1 64.537} C_DIS
LIN {X 0.092,Y -575.054,Z 709.154,A 0.000,B 0.000,C 90.000,E1 63.691} C_DIS
LIN {X 0.144,Y -572.879,Z 709.149,A 0.000,B 0.000,C 90.000,E1 62.871} C_DIS
LIN {X -0.341,Y -570.498,Z 709.145,A 0.000,B 0.000,C 90.000,E1 62.103} C_DIS
LIN {X 0.019,Y -567.084,Z 709.139,A 0.000,B 0.000,C 90.000,E1 60.973} C_DIS
LIN {X 0.244,Y -564.262,Z 709.134,A 0.000,B 0.000,C 90.000,E1 60.127} C_DIS
LIN {X -0.053,Y -561.225,Z 709.130,A 0.000,B 0.000,C 90.000,E1 59.331} C_DIS
LIN {X 0.095,Y -557.796,Z 709.125,A 0.000,B 0.000,C 90.000,E1 58.486} C_DIS
LIN {X 0.131,Y -554.653,Z 709.121,A 0.000,B 0.000,C 90.000,E1 57.788} C_DIS
LIN {X -0.155,Y -551.113,Z 709.117,A 0.000,B 0.000,C 90.000,E1 57.120} C_DIS
LIN {X -0.300,Y -546.254,Z 709.113,A 0.000,B 0.000,C 90.000,E1 56.294} C_DIS
LIN {X 0.364,Y -543.719,Z 709.110,A 0.000,B 0.000,C 90.000,E1 55.801} C_DIS
LIN {X 0.281,Y -539.036,Z 709.106,A 0.000,B 0.000,C 90.000,E1 55.102} C_DIS
LIN {X 0.000,Y -534.979,Z 709.103,A 0.000,B 0.000,C 90.000,E1 54.562} C_DIS
LIN {X 0.000,Y -530.383,Z 709.100,A 0.000,B 0.000,C 90.000,E1 53.989} C_DIS
LIN {X 0.135,Y -526.673,Z 709.098,A 0.000,B 0.000,C 90.000,E1 53.543} C_DIS
LIN {X -0.059,Y -521.326,Z 709.094,A 0.000,B 0.000,C 90.000,E1 53.004} C_DIS
LIN {X 0.038,Y -515.654,Z 709.092,A 0.000,B 0.000,C 90.000,E1 52.477} C_DIS
LIN {X 0.019,Y -511.144,Z 709.090,A 0.000,B 0.000,C 90.000,E1 52.110} C_DIS
LIN {X 0.170,Y -504.776,Z 709.087,A 0.000,B 0.000,C 90.000,E1 51.618} C_DIS
LIN {X 0.256,Y -498.271,Z 709.084,A 0.000,B 0.000,C 90.000,E1 51.170} C_DIS
LIN {X 0.029,Y -490.132,Z 709.082,A 0.000,B 0.000,C 90.000,E1 50.678} C_DIS
LIN {X -0.177,Y -475.354,Z 709.077,A 0.000,B 0.000,C 90.000,E1 49.828} C_DIS
LIN {X 0.112,Y -455.702,Z 709.070,A 0.000,B 0.000,C 90.000,E1 48.609} C_DIS
LIN {X 0.111,Y -442.663,Z 709.066,A 0.000,B 0.000,C 90.000,E1 47.796} C_DIS
LIN {X -0.082,Y -436.086,Z 709.063,A 0.000,B 0.000,C 90.000,E1 47.391} C_DIS
LIN {X 0.171,Y -432.785,Z 709.062,A 0.000,B 0.000,C 90.000,E1 47.148} C_DIS
LIN {X -0.037,Y -421.384,Z 709.057,A 0.000,B 0.000,C 90.000,E1 46.338} C_DIS
LIN {X 0.241,Y -421.374,Z 709.057,A 0.000,B 0.000,C 90.000,E1 46.296} C_DIS
LIN {X 0.049,Y -418.824,Z 709.050,A 0.000,B 0.000,C 90.000,E1 44.919} C_DIS
LIN {X 0.174,Y -415.645,Z 709.042,A 0.000,B 0.000,C 90.000,E1 43.542} C_DIS
LIN {X 0.001,Y -408.637,Z 709.023,A 0.000,B 0.000,C 90.000,E1 40.135} C_DIS
LIN {X 0.046,Y -408.540,Z 709.019,A 0.000,B 0.000,C 90.000,E1 39.439} C_DIS
LIN {X -0.028,Y -408.830,Z 709.006,A 0.000,B 0.000,C 90.000,E1 37.030} C_DIS
LIN {X 0.053,Y -409.908,Z 708.988,A 0.000,B 0.000,C 90.000,E1 33.913} C_DIS
LIN {X -0.043,Y -411.035,Z 708.975,A 0.000,B 0.000,C 90.000,E1 31.514} C_DIS
LIN {X -0.051,Y -411.900,Z 708.966,A 0.000,B 0.000,C 90.000,E1 29.795} C_DIS
LIN {X -0.237,Y -412.892,Z 708.956,A 0.000,B 0.000,C 90.000,E1 28.103} C_DIS
LIN {X -0.056,Y -414.655,Z 708.941,A 0.000,B 0.000,C 90.000,E1 25.335} C_DIS
LIN {X 0.127,Y -416.260,Z 708.929,A 0.000,B 0.000,C 90.000,E1 23.259} C_DIS
LIN {X -0.046,Y -418.733,Z 708.914,A 0.000,B 0.000,C 90.000,E1 20.556} C_DIS
LIN {X -0.003,Y -420.513,Z 708.905,A 0.000,B 0.000,C 90.000,E1 18.852} C_DIS
LIN {X 0.119,Y -422.762,Z 708.893,A 0.000,B 0.000,C 90.000,E1 16.804} C_DIS
LIN {X 0.170,Y -425.243,Z 708.882,A 0.000,B 0.000,C 90.000,E1 14.773} C_DIS
LIN {X 0.063,Y -427.824,Z 708.871,A 0.000,B 0.000,C 90.000,E1 12.771} C_DIS
LIN {X -0.181,Y -430.099,Z 708.862,A 0.000,B 0.000,C 90.000,E1 11.130} C_DIS
LIN {X -0.226,Y -433.225,Z 708.849,A 0.000,B 0.000,C 90.000,E1 8.803} C_DIS
LIN {X 0.042,Y -436.043,Z 708.838,A 0.000,B 0.000,C 90.000,E1 6.777} C_DIS
LIN {X -0.017,Y -439.372,Z 708.825,A 0.000,B 0.000,C 90.000,E1 4.473} C_DIS
LIN {X -0.049,Y -443.036,Z 708.812,A 0.000,B 0.000,C 90.000,E1 2.178} C_DIS
LIN {X 0.000,Y -446.792,Z 708.800,A 0.000,B 0.000,C 90.000,E1 360.000} C_DIS
LIN {X 0.030,Y -450.251,Z 708.790,A 0.000,B 0.000,C 90.000,E1 358.165} C_DIS
LIN {X 0.031,Y -455.356,Z 708.776,A 0.000,B 0.000,C 90.000,E1 355.584} C_DIS
LIN {X -0.164,Y -459.282,Z 708.765,A 0.000,B 0.000,C 90.000,E1 353.685} C_DIS
LIN {X 0.052,Y -462.558,Z 708.756,A 0.000,B 0.000,C 90.000,E1 352.064} C_DIS
LIN {X 0.139,Y -466.285,Z 708.745,A 0.000,B 0.000,C 90.000,E1 350.151} C_DIS
LIN {X -0.163,Y -468.731,Z 708.738,A 0.000,B 0.000,C 90.000,E1 348.926} C_DIS
LIN {X -0.152,Y -471.557,Z 708.730,A 0.000,B 0.000,C 90.000,E1 347.353} C_DIS
LIN {X -0.050,Y -474.997,Z 708.719,A 0.000,B 0.000,C 90.000,E1 345.463} C_DIS
LIN {X 0.031,Y -476.741,Z 708.714,A 0.000,B 0.000,C 90.000,E1 344.519} C_DIS
LIN {X 0.076,Y -479.680,Z 708.705,A 0.000,B 0.000,C 90.000,E1 342.960} C_DIS
LIN {X 0.020,Y -484.692,Z 708.692,A 0.000,B 0.000,C 90.000,E1 340.496} C_DIS
LIN {X 0.103,Y -488.658,Z 708.681,A 0.000,B 0.000,C 90.000,E1 338.646} C_DIS
LIN {X 0.155,Y -490.293,Z 708.678,A 0.000,B 0.000,C 90.000,E1 338.028} C_DIS
LIN {X -0.026,Y -491.831,Z 708.676,A 0.000,B 0.000,C 90.000,E1 337.592} C_DIS
LIN {X 0.257,Y -493.980,Z 708.673,A 0.000,B 0.000,C 90.000,E1 337.102} C_DIS
LIN {X 0.063,Y -496.123,Z 708.671,A 0.000,B 0.000,C 90.000,E1 336.794} C_DIS
LIN {X 0.182,Y -498.656,Z 708.670,A 0.000,B 0.000,C 90.000,E1 336.485} C_DIS
LIN {X -0.077,Y -503.558,Z 708.667,A 0.000,B 0.000,C 90.000,E1 336.049} C_DIS
LIN {X -0.025,Y -509.170,Z 708.665,A 0.000,B 0.000,C 90.000,E1 335.613} C_DIS
LIN {X -0.260,Y -529.566,Z 708.657,A 0.000,B 0.000,C 90.000,E1 334.280} C_DIS
LIN {X 0.022,Y -537.281,Z 708.654,A 0.000,B 0.000,C 90.000,E1 333.717} C_DIS
LIN {X 0.107,Y -541.820,Z 708.652,A 0.000,B 0.000,C 90.000,E1 333.384} C_DIS
LIN {X 0.050,Y -546.275,Z 708.650,A 0.000,B 0.000,C 90.000,E1 333.050} C_DIS
LIN {X -0.285,Y -552.052,Z 708.648,A 0.000,B 0.000,C 90.000,E1 332.615} C_DIS
LIN {X 0.050,Y -560.205,Z 708.644,A 0.000,B 0.000,C 90.000,E1 331.847} C_DIS
LIN {X -0.322,Y -566.654,Z 708.640,A 0.000,B 0.000,C 90.000,E1 331.257} C_DIS
LIN {X -0.169,Y -572.902,Z 708.637,A 0.000,B 0.000,C 90.000,E1 330.589} C_DIS
LIN {X -0.051,Y -580.223,Z 708.632,A 0.000,B 0.000,C 90.000,E1 329.793} C_DIS
LIN {X -0.104,Y -589.452,Z 708.626,A 0.000,B 0.000,C 90.000,E1 328.742} C_DIS
LIN {X 0.124,Y -597.454,Z 708.621,A 0.000,B 0.000,C 90.000,E1 327.788} C_DIS
LIN {X 0.171,Y -603.963,Z 708.617,A 0.000,B 0.000,C 90.000,E1 326.993} C_DIS
LIN {X 0.106,Y -609.942,Z 708.612,A 0.000,B 0.000,C 90.000,E1 326.215} C_DIS
LIN {X -0.240,Y -615.657,Z 708.608,A 0.000,B 0.000,C 90.000,E1 325.468} C_DIS
LIN {X -0.160,Y -620.116,Z 708.604,A 0.000,B 0.000,C 90.000,E1 324.815} C_DIS
LIN {X -0.050,Y -625.167,Z 708.600,A 0.000,B 0.000,C 90.000,E1 324.036} C_DIS
LIN {X 0.113,Y -629.953,Z 708.596,A 0.000,B 0.000,C 90.000,E1 323.256} C_DIS
LIN {X -0.191,Y -635.887,Z 708.590,A 0.000,B 0.000,C 90.000,E1 322.271} C_DIS
LIN {X -0.133,Y -642.923,Z 708.583,A 0.000,B 0.000,C 90.000,E1 321.009} C_DIS
LIN {X 0.117,Y -648.228,Z 708.578,A 0.000,B 0.000,C 90.000,E1 319.989} C_DIS
LIN {X -0.063,Y -653.250,Z 708.572,A 0.000,B 0.000,C 90.000,E1 319.013} C_DIS
LIN {X -0.232,Y -658.572,Z 708.566,A 0.000,B 0.000,C 90.000,E1 317.919} C_DIS
LIN {X 0.172,Y -661.845,Z 708.562,A 0.000,B 0.000,C 90.000,E1 317.148} C_DIS
LIN {X -0.340,Y -665.990,Z 708.557,A 0.000,B 0.000,C 90.000,E1 316.215} C_DIS
LIN {X -0.346,Y -668.794,Z 708.553,A 0.000,B 0.000,C 90.000,E1 315.486} C_DIS
LIN {X -0.273,Y -674.146,Z 708.544,A 0.000,B 0.000,C 90.000,E1 314.028} C_DIS
LIN {X 0.389,Y -679.007,Z 708.536,A 0.000,B 0.000,C 90.000,E1 312.528} C_DIS
LIN {X 0.089,Y -682.170,Z 708.531,A 0.000,B 0.000,C 90.000,E1 311.595} C_DIS
LIN {X 0.340,Y -685.027,Z 708.526,A 0.000,B 0.000,C 90.000,E1 310.620} C_DIS
LIN {X -0.336,Y -687.671,Z 708.521,A 0.000,B 0.000,C 90.000,E1 309.725} C_DIS
LIN {X -0.388,Y -690.491,Z 708.514,A 0.000,B 0.000,C 90.000,E1 308.543} C_DIS
LIN {X -0.038,Y -692.365,Z 708.509,A 0.000,B 0.000,C 90.000,E1 307.569} C_DIS
LIN {X -0.095,Y -694.016,Z 708.503,A 0.000,B 0.000,C 90.000,E1 306.629} C_DIS
LIN {X -0.191,Y -695.167,Z 708.500,A 0.000,B 0.000,C 90.000,E1 305.931} C_DIS
LIN {X -0.049,Y -696.476,Z 708.494,A 0.000,B 0.000,C 90.000,E1 304.978} C_DIS
LIN {X 0.171,Y -697.890,Z 708.488,A 0.000,B 0.000,C 90.000,E1 303.785} C_DIS
LIN {X -0.225,Y -698.841,Z 708.483,A 0.000,B 0.000,C 90.000,E1 302.880} C_DIS
LIN {X 0.151,Y -700.267,Z 708.474,A 0.000,B 0.000,C 90.000,E1 301.209} C_DIS
LIN {X -0.259,Y -700.743,Z 708.470,A 0.000,B 0.000,C 90.000,E1 300.541} C_DIS
LIN {X -0.049,Y -701.138,Z 708.464,A 0.000,B 0.000,C 90.000,E1 299.589} C_DIS
LIN {X -0.041,Y -701.718,Z 708.454,A 0.000,B 0.000,C 90.000,E1 297.719} C_DIS
LIN {X 0.271,Y -702.701,Z 708.442,A 0.000,B 0.000,C 90.000,E1 295.591} C_DIS
LIN {X -0.105,Y -702.819,Z 708.440,A 0.000,B 0.000,C 90.000,E1 295.155} C_DIS
LIN {X -0.183,Y -702.267,Z 708.437,A 0.000,B 0.000,C 90.000,E1 294.695} C_DIS
LIN {X -0.197,Y -701.891,Z 708.436,A 0.000,B 0.000,C 90.000,E1 294.463} C_DIS
LIN {X 0.080,Y -700.831,Z 708.435,A 0.000,B 0.000,C 90.000,E1 294.207} C_DIS
LIN {X -0.151,Y -698.895,Z 708.433,A 0.000,B 0.000,C 90.000,E1 293.875} C_DIS
LIN {X -0.300,Y -698.121,Z 708.432,A 0.000,B 0.000,C 90.000,E1 293.770} C_DIS
LIN {X -0.167,Y -696.968,Z 708.431,A 0.000,B 0.000,C 90.000,E1 293.643} C_DIS
LIN {X -0.036,Y -695.265,Z 708.431,A 0.000,B 0.000,C 90.000,E1 293.515} C_DIS
LIN {X 0.180,Y -688.772,Z 708.429,A 0.000,B 0.000,C 90.000,E1 293.131} C_DIS
LIN {X -0.180,Y -686.443,Z 708.428,A 0.000,B 0.000,C 90.000,E1 293.078} C_DIS
LIN {X -0.309,Y -677.379,Z 708.427,A 0.000,B 0.000,C 90.000,E1 292.898} C_DIS
LIN {X 0.067,Y -663.396,Z 708.426,A 0.000,B 0.000,C 90.000,E1 292.695} C_DIS
LIN {X -0.297,Y -646.079,Z 708.425,A 0.000,B 0.000,C 90.000,E1 292.461} C_DIS
LIN {X -0.095,Y -636.315,Z 708.424,A 0.000,B 0.000,C 90.000,E1 292.259} C_DIS
LIN {X -0.069,Y -623.059,Z 708.422,A 0.000,B 0.000,C 90.000,E1 291.950} C_DIS
LIN {X 0.253,Y -606.003,Z 708.419,A 0.000,B 0.000,C 90.000,E1 291.461} C_DIS
LIN {X -0.057,Y -578.171,Z 708.415,A 0.000,B 0.000,C 90.000,E1 290.663} C_DIS
LIN {X -0.316,Y -569.132,Z 708.413,A 0.000,B 0.000,C 90.000,E1 290.429} C_DIS
LIN {X 0.163,Y -562.049,Z 708.412,A 0.000,B 0.000,C 90.000,E1 290.120} C_DIS
LIN {X 0.237,Y -559.394,Z 708.411,A 0.000,B 0.000,C 90.000,E1 289.993} C_DIS
LIN {X -0.234,Y -556.087,Z 708.410,A 0.000,B 0.000,C 90.000,E1 289.812} C_DIS
LIN {X 0.252,Y -556.036,Z 708.410,A 0.000,B 0.000,C 90.000,E1 289.758} C_DIS
LIN {X -0.011,Y -555.380,Z 708.409,A 0.000,B 0.000,C 90.000,E1 289.631} C_DIS
LIN {X -0.129,Y -555.113,Z 708.408,A 0.000,B 0.000,C 90.000,E1 289.504} C_DIS
LIN {X -0.026,Y -554.776,Z 708.407,A 0.000,B 0.000,C 90.000,E1 289.214} C_DIS
LIN {X -0.159,Y -553.886,Z 708.396,A 0.000,B 0.000,C 90.000,E1 287.275} C_DIS
LIN {X 0.191,Y -553.375,Z 708.388,A 0.000,B 0.000,C 90.000,E1 285.843} C_DIS
LIN {X 0.224,Y -552.695,Z 708.377,A 0.000,B 0.000,C 90.000,E1 283.883} C_DIS
LIN {X -0.019,Y -551.997,Z 708.366,A 0.000,B 0.000,C 90.000,E1 281.951} C_DIS
LIN {X 0.030,Y -551.366,Z 708.359,A 0.000,B 0.000,C 90.000,E1 280.546} C_DIS
LIN {X 0.080,Y -550.547,Z 708.349,A 0.000,B 0.000,C 90.000,E1 278.859} C_DIS
LIN {X 0.130,Y -549.791,Z 708.338,A 0.000,B 0.000,C 90.000,E1 276.891} C_DIS
LIN {X 0.169,Y -549.181,Z 708.324,A 0.000,B 0.000,C 90.000,E1 274.359} C_DIS
LIN {X -0.074,Y -548.808,Z 708.317,A 0.000,B 0.000,C 90.000,E1 272.980} C_DIS
LIN {X 0.238,Y -548.275,Z 708.307,A 0.000,B 0.000,C 90.000,E1 271.260} C_DIS
LIN {X -0.114,Y -547.732,Z 708.301,A 0.000,B 0.000,C 90.000,E1 270.172} C_DIS
LIN {X 0.205,Y -546.501,Z 708.290,A 0.000,B 0.000,C 90.000,E1 268.167} C_DIS
LIN {X -0.093,Y -545.700,Z 708.282,A 0.000,B 0.000,C 90.000,E1 266.788} C_DIS
LIN {X 0.112,Y -544.673,Z 708.274,A 0.000,B 0.000,C 90.000,E1 265.355} C_DIS
LIN {X -0.138,Y -543.451,Z 708.265,A 0.000,B 0.000,C 90.000,E1 263.685} C_DIS
LIN {X 0.038,Y -542.473,Z 708.259,A 0.000,B 0.000,C 90.000,E1 262.534} C_DIS
LIN {X -0.116,Y -540.936,Z 708.249,A 0.000,B 0.000,C 90.000,E1 260.849} C_DIS
LIN {X 0.165,Y -539.662,Z 708.241,A 0.000,B 0.000,C 90.000,E1 259.398} C_DIS
LIN {X 0.125,Y -537.833,Z 708.230,A 0.000,B 0.000,C 90.000,E1 257.409} C_DIS
LIN {X 0.150,Y -535.960,Z 708.219,A 0.000,B 0.000,C 90.000,E1 255.408} C_DIS
LIN {X -0.025,Y -534.869,Z 708.213,A 0.000,B 0.000,C 90.000,E1 254.283} C_DIS
LIN {X -0.031,Y -533.436,Z 708.205,A 0.000,B 0.000,C 90.000,E1 252.851} C_DIS
LIN {X 0.095,Y -531.979,Z 708.197,A 0.000,B 0.000,C 90.000,E1 251.402} C_DIS
LIN {X 0.184,Y -530.749,Z 708.190,A 0.000,B 0.000,C 90.000,E1 250.242} C_DIS
LIN {X -0.058,Y -528.471,Z 708.181,A 0.000,B 0.000,C 90.000,E1 248.539} C_DIS
LIN {X 0.171,Y -526.810,Z 708.174,A 0.000,B 0.000,C 90.000,E1 247.358} C_DIS
LIN {X -0.103,Y -525.156,Z 708.168,A 0.000,B 0.000,C 90.000,E1 246.230} C_DIS
LIN {X 0.137,Y -522.255,Z 708.158,A 0.000,B 0.000,C 90.000,E1 244.460} C_DIS
LIN {X 0.114,Y -520.767,Z 708.153,A 0.000,B 0.000,C 90.000,E1 243.589} C_DIS
LIN {X 0.210,Y -518.551,Z 708.147,A 0.000,B 0.000,C 90.000,E1 242.410} C_DIS
LIN {X -0.053,Y -515.682,Z 708.139,A 0.000,B 0.000,C 90.000,E1 240.973} C_DIS
LIN {X 0.072,Y -512.639,Z 708.131,A 0.000,B 0.000,C 90.000,E1 239.488} C_DIS
LIN {X 0.211,Y -509.494,Z 708.122,A 0.000,B 0.000,C 90.000,E1 237.995} C_DIS
LIN {X -0.126,Y -506.359,Z 708.114,A 0.000,B 0.000,C 90.000,E1 236.548} C_DIS
LIN {X -0.102,Y -503.182,Z 708.106,A 0.000,B 0.000,C 90.000,E1 235.055} C_DIS
LIN {X -0.034,Y -501.202,Z 708.101,A 0.000,B 0.000,C 90.000,E1 234.149} C_DIS
LIN {X 0.180,Y -498.151,Z 708.094,A 0.000,B 0.000,C 90.000,E1 232.924} C_DIS
LIN {X -0.176,Y -494.328,Z 708.086,A 0.000,B 0.000,C 90.000,E1 231.457} C_DIS
LIN {X 0.094,Y -489.117,Z 708.074,A 0.000,B 0.000,C 90.000,E1 229.299} C_DIS
LIN {X 0.063,Y -486.292,Z 708.067,A 0.000,B 0.000,C 90.000,E1 228.081} C_DIS
LIN {X -0.289,Y -481.413,Z 708.055,A 0.000,B 0.000,C 90.000,E1 225.972} C_DIS
LIN {X -0.101,Y -476.659,Z 708.043,A 0.000,B 0.000,C 90.000,E1 223.785} C_DIS
LIN {X 0.054,Y -471.192,Z 708.029,A 0.000,B 0.000,C 90.000,E1 221.272} C_DIS
LIN {X -0.055,Y -467.226,Z 708.019,A 0.000,B 0.000,C 90.000,E1 219.402} C_DIS
LIN {X 0.062,Y -463.757,Z 708.010,A 0.000,B 0.000,C 90.000,E1 217.810} C_DIS
LIN {X -0.143,Y -459.669,Z 708.000,A 0.000,B 0.000,C 90.000,E1 215.931} C_DIS
LIN {X 0.089,Y -457.747,Z 707.994,A 0.000,B 0.000,C 90.000,E1 214.945} C_DIS
LIN {X 0.037,Y -455.960,Z 707.989,A 0.000,B 0.000,C 90.000,E1 213.992} C_DIS
LIN {X -0.019,Y -451.679,Z 707.976,A 0.000,B 0.000,C 90.000,E1 211.750} C_DIS
LIN {X 0.038,Y -446.902,Z 707.962,A 0.000,B 0.000,C 90.000,E1 209.155} C_DIS
LIN {X 0.002,Y -443.370,Z 707.951,A 0.000,B 0.000,C 90.000,E1 207.206} C_DIS
LIN {X 0.266,Y -439.803,Z 707.940,A 0.000,B 0.000,C 90.000,E1 205.207} C_DIS
LIN {X 0.060,Y -436.167,Z 707.929,A 0.000,B 0.000,C 90.000,E1 203.259} C_DIS
LIN {X -0.042,Y -434.362,Z 707.924,A 0.000,B 0.000,C 90.000,E1 202.280} C_DIS
LIN {X -0.138,Y -430.728,Z 707.913,A 0.000,B 0.000,C 90.000,E1 200.301} C_DIS
LIN {X -0.080,Y -427.098,Z 707.902,A 0.000,B 0.000,C 90.000,E1 198.290} C_DIS
LIN {X 0.214,Y -422.808,Z 707.889,A 0.000,B 0.000,C 90.000,E1 195.898} C_DIS
LIN {X 0.108,Y -419.100,Z 707.877,A 0.000,B 0.000,C 90.000,E1 193.883} C_DIS
LIN {X -0.136,Y -414.933,Z 707.864,A 0.000,B 0.000,C 90.000,E1 191.535} C_DIS
LIN {X 0.089,Y -412.017,Z 707.854,A 0.000,B 0.000,C 90.000,E1 189.792} C_DIS
LIN {X -0.132,Y -407.663,Z 707.839,A 0.000,B 0.000,C 90.000,E1 187.068} C_DIS
LIN {X -0.150,Y -404.539,Z 707.828,A 0.000,B 0.000,C 90.000,E1 184.992} C_DIS
LIN {X 0.073,Y -401.158,Z 707.814,A 0.000,B 0.000,C 90.000,E1 182.522} C_DIS
LIN {X 0.162,Y -398.279,Z 707.800,A 0.000,B 0.000,C 90.000,E1 180.057} C_DIS
LIN {X -0.075,Y -394.544,Z 707.779,A 0.000,B 0.000,C 90.000,E1 176.216} C_DIS
LIN {X 0.068,Y -392.093,Z 707.757,A 0.000,B 0.000,C 90.000,E1 172.299} C_DIS
LIN {X 0.182,Y -391.140,Z 707.745,A 0.000,B 0.000,C 90.000,E1 170.151} C_DIS
LIN {X -0.094,Y -390.351,Z 707.732,A 0.000,B 0.000,C 90.000,E1 167.701} C_DIS
LIN {X 0.211,Y -389.712,Z 707.720,A 0.000,B 0.000,C 90.000,E1 165.519} C_DIS
LIN {X -0.224,Y -389.258,Z 707.706,A 0.000,B 0.000,C 90.000,E1 163.087} C_DIS
LIN {X 0.039,Y -389.090,Z 707.692,A 0.000,B 0.000,C 90.000,E1 160.550} C_DIS
LIN {X 0.024,Y -389.027,Z 707.680,A 0.000,B 0.000,C 90.000,E1 158.411} C_DIS
LIN {X -0.058,Y -389.162,Z 707.668,A 0.000,B 0.000,C 90.000,E1 156.282} C_DIS
LIN {X 0.053,Y -389.445,Z 707.654,A 0.000,B 0.000,C 90.000,E1 153.768} C_DIS
LIN {X -0.065,Y -389.634,Z 707.646,A 0.000,B 0.000,C 90.000,E1 152.359} C_DIS
LIN {X 0.146,Y -390.573,Z 707.625,A 0.000,B 0.000,C 90.000,E1 148.408} C_DIS
LIN {X -0.001,Y -391.658,Z 707.613,A 0.000,B 0.000,C 90.000,E1 146.294} C_DIS
LIN {X -0.122,Y -394.340,Z 707.593,A 0.000,B 0.000,C 90.000,E1 142.763} C_DIS
LIN {X 0.180,Y -397.784,Z 707.575,A 0.000,B 0.000,C 90.000,E1 139.542} C_DIS
LIN {X -0.087,Y -400.563,Z 707.564,A 0.000,B 0.000,C 90.000,E1 137.472} C_DIS
LIN {X 0.021,Y -401.191,Z 707.562,A 0.000,B 0.000,C 90.000,E1 137.106} C_DIS
LIN {X 0.136,Y -403.325,Z 707.557,A 0.000,B 0.000,C 90.000,E1 136.215} C_DIS
LIN {X 0.020,Y -405.493,Z 707.554,A 0.000,B 0.000,C 90.000,E1 135.688} C_DIS
LIN {X 0.220,Y -406.387,Z 707.553,A 0.000,B 0.000,C 90.000,E1 135.486} C_DIS
LIN {X -0.005,Y -409.759,Z 707.550,A 0.000,B 0.000,C 90.000,E1 135.000} C_DIS
LIN {X -0.021,Y -412.754,Z 707.548,A 0.000,B 0.000,C 90.000,E1 134.636} C_DIS
LIN {X 0.150,Y -422.344,Z 707.543,A 0.000,B 0.000,C 90.000,E1 133.623} C_DIS
LIN {X 0.158,Y -437.499,Z 707.535,A 0.000,B 0.000,C 90.000,E1 132.204} C_DIS
LIN {X -0.135,Y -448.146,Z 707.529,A 0.000,B 0.000,C 90.000,E1 131.310} C_DIS
LIN {X -0.089,Y -460.335,Z 707.524,A 0.000,B 0.000,C 90.000,E1 130.253} C_DIS
LIN {X 0.084,Y -469.251,Z 707.519,A 0.000,B 0.000,C 90.000,E1 129.439} C_DIS
LIN {X 0.246,Y -476.530,Z 707.516,A 0.000,B 0.000,C 90.000,E1 128.749} C_DIS
LIN {X -0.080,Y -487.908,Z 707.509,A 0.000,B 0.000,C 90.000,E1 127.684} C_DIS
LIN {X 0.211,Y -494.721,Z 707.505,A 0.000,B 0.000,C 90.000,E1 126.950} C_DIS
LIN {X 0.061,Y -501.488,Z 707.501,A 0.000,B 0.000,C 90.000,E1 126.251} C_DIS
LIN {X -0.213,Y -506.481,Z 707.498,A 0.000,B 0.000,C 90.000,E1 125.724} C_DIS
LIN {X 0.239,Y -511.215,Z 707.495,A 0.000,B 0.000,C 90.000,E1 125.105} C_DIS
LIN {X 0.026,Y -515.592,Z 707.492,A 0.000,B 0.000,C 90.000,E1 124.565} C_DIS
LIN {X -0.114,Y -519.822,Z 707.489,A 0.000,B 0.000,C 90.000,E1 123.992} C_DIS
LIN {X -0.136,Y -524.434,Z 707.485,A 0.000,B 0.000,C 90.000,E1 123.293} C_DIS
LIN {X 0.116,Y -527.935,Z 707.482,A 0.000,B 0.000,C 90.000,E1 122.704} C_DIS
LIN {X -0.104,Y -532.027,Z 707.478,A 0.000,B 0.000,C 90.000,E1 122.005} C_DIS
LIN {X 0.162,Y -535.732,Z 707.474,A 0.000,B 0.000,C 90.000,E1 121.258} C_DIS
LIN {X 0.187,Y -539.153,Z 707.470,A 0.000,B 0.000,C 90.000,E1 120.541} C_DIS
LIN {X -0.004,Y -544.729,Z 707.463,A 0.000,B 0.000,C 90.000,E1 119.283} C_DIS
LIN {X 0.120,Y -548.755,Z 707.457,A 0.000,B 0.000,C 90.000,E1 118.281} C_DIS
LIN {X -0.112,Y -552.015,Z 707.453,A 0.000,B 0.000,C 90.000,E1 117.462} C_DIS
LIN {X -0.052,Y -555.083,Z 707.448,A 0.000,B 0.000,C 90.000,E1 116.616} C_DIS
LIN {X 0.325,Y -558.844,Z 707.442,A 0.000,B 0.000,C 90.000,E1 115.463} C_DIS
LIN {X 0.210,Y -561.336,Z 707.437,A 0.000,B 0.000,C 90.000,E1 114.643} C_DIS
LIN {X -0.078,Y -564.177,Z 707.431,A 0.000,B 0.000,C 90.000,E1 113.567} C_DIS
LIN {X -0.173,Y -565.467,Z 707.428,A 0.000,B 0.000,C 90.000,E1 113.025} C_DIS
LIN {X -0.034,Y -566.634,Z 707.425,A 0.000,B 0.000,C 90.000,E1 112.461} C_DIS
LIN {X -0.134,Y -569.086,Z 707.417,A 0.000,B 0.000,C 90.000,E1 111.099} C_DIS
LIN {X -0.016,Y -570.913,Z 707.411,A 0.000,B 0.000,C 90.000,E1 109.993} C_DIS
LIN {X -0.080,Y -573.649,Z 707.402,A 0.000,B 0.000,C 90.000,E1 108.362} C_DIS
LIN {X -0.091,Y -575.326,Z 707.396,A 0.000,B 0.000,C 90.000,E1 107.275} C_DIS
LIN {X 0.115,Y -577.385,Z 707.388,A 0.000,B 0.000,C 90.000,E1 105.898} C_DIS
LIN {X 0.201,Y -579.377,Z 707.381,A 0.000,B 0.000,C 90.000,E1 104.537} C_DIS
LIN {X 0.320,Y -581.315,Z 707.373,A 0.000,B 0.000,C 90.000,E1 103.175} C_DIS
LIN {X -0.206,Y -584.432,Z 707.361,A 0.000,B 0.000,C 90.000,E1 101.074} C_DIS
LIN {X -0.138,Y -586.363,Z 707.354,A 0.000,B 0.000,C 90.000,E1 99.726} C_DIS
LIN {X 0.180,Y -587.660,Z 707.348,A 0.000,B 0.000,C 90.000,E1 98.624} C_DIS
LIN {X -0.297,Y -589.616,Z 707.339,A 0.000,B 0.000,C 90.000,E1 97.068} C_DIS
LIN {X 0.114,Y -591.695,Z 707.329,A 0.000,B 0.000,C 90.000,E1 95.163} C_DIS
LIN {X 0.047,Y -593.154,Z 707.321,A 0.000,B 0.000,C 90.000,E1 93.841} C_DIS
LIN {X -0.252,Y -594.154,Z 707.315,A 0.000,B 0.000,C 90.000,E1 92.808} C_DIS
LIN {X 0.054,Y -595.069,Z 707.310,A 0.000,B 0.000,C 90.000,E1 91.718} C_DIS
LIN {X -0.239,Y -595.848,Z 707.304,A 0.000,B 0.000,C 90.000,E1 90.688} C_DIS
LIN {X -0.151,Y -596.367,Z 707.299,A 0.000,B 0.000,C 90.000,E1 89.885} C_DIS
LIN {X 0.173,Y -596.823,Z 707.293,A 0.000,B 0.000,C 90.000,E1 88.797} C_DIS
LIN {X 0.153,Y -597.285,Z 707.286,A 0.000,B 0.000,C 90.000,E1 87.478} C_DIS
LIN {X 0.139,Y -597.605,Z 707.279,A 0.000,B 0.000,C 90.000,E1 86.159} C_DIS
LIN {X 0.169,Y -597.817,Z 707.271,A 0.000,B 0.000,C 90.000,E1 84.837} C_DIS
LIN {X 0.200,Y -597.783,Z 707.264,A 0.000,B 0.000,C 90.000,E1 83.514} C_DIS
LIN {X -0.009,Y -597.596,Z 707.255,A 0.000,B 0.000,C 90.000,E1 81.951} C_DIS
LIN {X -0.115,Y -597.232,Z 707.249,A 0.000,B 0.000,C 90.000,E1 80.905} C_DIS
LIN {X -0.223,Y -596.687,Z 707.244,A 0.000,B 0.000,C 90.000,E1 79.859} C_DIS
LIN {X -0.055,Y -595.867,Z 707.236,A 0.000,B 0.000,C 90.000,E1 78.522} C_DIS
LIN {X 0.212,Y -594.846,Z 707.229,A 0.000,B 0.000,C 90.000,E1 77.173} C_DIS
LIN {X 0.177,Y -593.960,Z 707.223,A 0.000,B 0.000,C 90.000,E1 76.117} C_DIS
LIN {X 0.274,Y -592.982,Z 707.217,A 0.000,B 0.000,C 90.000,E1 75.046} C_DIS
LIN {X 0.054,Y -591.677,Z 707.210,A 0.000,B 0.000,C 90.000,E1 73.740} C_DIS
LIN {X 0.091,Y -589.587,Z 707.199,A 0.000,B 0.000,C 90.000,E1 71.873} C_DIS
LIN {X 0.305,Y -588.226,Z 707.193,A 0.000,B 0.000,C 90.000,E1 70.786} C_DIS
LIN {X 0.156,Y -586.387,Z 707.186,A 0.000,B 0.000,C 90.000,E1 69.464} C_DIS
LIN {X -0.162,Y -584.342,Z 707.179,A 0.000,B 0.000,C 90.000,E1 68.156} C_DIS
LIN {X -0.103,Y -583.476,Z 707.176,A 0.000,B 0.000,C 90.000,E1 67.614} C_DIS
LIN {X -0.097,Y -581.501,Z 707.170,A 0.000,B 0.000,C 90.000,E1 66.538} C_DIS
LIN {X -0.347,Y -579.284,Z 707.164,A 0.000,B 0.000,C 90.000,E1 65.485} C_DIS
LIN {X -0.247,Y -577.414,Z 707.159,A 0.000,B 0.000,C 90.000,E1 64.665} C_DIS
LIN {X -0.066,Y -574.643,Z 707.153,A 0.000,B 0.000,C 90.000,E1 63.563} C_DIS
LIN {X -0.178,Y -571.620,Z 707.147,A 0.000,B 0.000,C 90.000,E1 62.487} C_DIS
LIN {X -0.076,Y -568.176,Z 707.141,A 0.000,B 0.000,C 90.000,E1 61.385} C_DIS
LIN {X -0.155,Y -566.417,Z 707.138,A 0.000,B 0.000,C 90.000,E1 60.845} C_DIS
LIN {X 0.062,Y -563.509,Z 707.133,A 0.000,B 0.000,C 90.000,E1 59.999} C_DIS
LIN {X -0.242,Y -560.350,Z 707.129,A 0.000,B 0.000,C 90.000,E1 59.203} C_DIS
LIN {X 0.003,Y -557.401,Z 707.125,A 0.000,B 0.000,C 90.000,E1 58.486} C_DIS
LIN {X 0.035,Y -554.150,Z 707.121,A 0.000,B 0.000,C 90.000,E1 57.788} C_DIS
LIN {X -0.257,Y -550.501,Z 707.117,A 0.000,B 0.000,C 90.000,E1 57.120} C_DIS
LIN {X 0.176,Y -546.415,Z 707.113,A 0.000,B 0.000,C 90.000,E1 56.373} C_DIS
LIN {X 0.253,Y -542.939,Z 707.110,A 0.000,B 0.000,C 90.000,E1 55.801} C_DIS
LIN {X 0.001,Y -539.129,Z 707.107,A 0.000,B 0.000,C 90.000,E1 55.261} C_DIS
LIN {X 0.029,Y -535.034,Z 707.104,A 0.000,B 0.000,C 90.000,E1 54.689} C_DIS
LIN {X 0.031,Y -530.411,Z 707.101,A 0.000,B 0.000,C 90.000,E1 54.116} C_DIS
LIN {X 0.054,Y -525.650,Z 707.098,A 0.000,B 0.000,C 90.000,E1 53.577} C_DIS
LIN {X 0.156,Y -520.538,Z 707.095,A 0.000,B 0.000,C 90.000,E1 53.050} C_DIS
LIN {X 0.207,Y -516.021,Z 707.093,A 0.000,B 0.000,C 90.000,E1 52.637} C_DIS
LIN {X -0.202,Y -509.889,Z 707.090,A 0.000,B 0.000,C 90.000,E1 52.190} C_DIS
LIN {X -0.050,Y -505.118,Z 707.088,A 0.000,B 0.000,C 90.000,E1 51.823} C_DIS
LIN {X 0.075,Y -498.627,Z 707.086,A 0.000,B 0.000,C 90.000,E1 51.376} C_DIS
LIN {X -0.131,Y -490.494,Z 707.083,A 0.000,B 0.000,C 90.000,E1 50.884} C_DIS
LIN {X -0.032,Y -474.097,Z 707.077,A 0.000,B 0.000,C 90.000,E1 49.908} C_DIS
LIN {X -0.014,Y -454.539,Z 707.071,A 0.000,B 0.000,C 90.000,E1 48.728} C_DIS
LIN {X 0.161,Y -440.066,Z 707.066,A 0.000,B 0.000,C 90.000,E1 47.796} C_DIS
LIN {X -0.059,Y -433.341,Z 707.063,A 0.000,B 0.000,C 90.000,E1 47.391} C_DIS
LIN {X 0.025,Y -421.816,Z 707.059,A 0.000,B 0.000,C 90.000,E1 46.539} C_DIS
LIN {X -0.002,Y -421.780,Z 707.059,A 0.000,B 0.000,C 90.000,E1 46.539} C_DIS
LIN {X 0.055,Y -418.605,Z 707.049,A 0.000,B 0.000,C 90.000,E1 44.798} C_DIS
LIN {X -0.141,Y -409.038,Z 707.024,A 0.000,B 0.000,C 90.000,E1 40.378} C_DIS
LIN {X 0.168,Y -408.924,Z 707.020,A 0.000,B 0.000,C 90.000,E1 39.644} C_DIS
LIN {X -0.054,Y -409.120,Z 707.009,A 0.000,B 0.000,C 90.000,E1 37.604} C_DIS
LIN {X 0.042,Y -410.110,Z 706.992,A 0.000,B 0.000,C 90.000,E1 34.485} C_DIS
LIN {X 0.111,Y -410.868,Z 706.982,A 0.000,B 0.000,C 90.000,E1 32.752} C_DIS
LIN {X -0.106,Y -411.947,Z 706.971,A 0.000,B 0.000,C 90.000,E1 30.718} C_DIS
LIN {X -0.065,Y -413.244,Z 706.957,A 0.000,B 0.000,C 90.000,E1 28.309} C_DIS
LIN {X 0.012,Y -414.729,Z 706.944,A 0.000,B 0.000,C 90.000,E1 25.899} C_DIS
LIN {X -0.046,Y -416.543,Z 706.931,A 0.000,B 0.000,C 90.000,E1 23.515} C_DIS
LIN {X -0.057,Y -419.006,Z 706.916,A 0.000,B 0.000,C 90.000,E1 20.791} C_DIS
LIN {X -0.070,Y -421.420,Z 706.902,A 0.000,B 0.000,C 90.000,E1 18.417} C_DIS
LIN {X 0.108,Y -422.971,Z 706.895,A 0.000,B 0.000,C 90.000,E1 17.040} C_DIS
LIN {X -0.172,Y -425.782,Z 706.882,A 0.000,B 0.000,C 90.000,E1 14.717} C_DIS
LIN {X -0.171,Y -428.353,Z 706.870,A 0.000,B 0.000,C 90.000,E1 12.703} C_DIS
LIN {X 0.007,Y -430.580,Z 706.861,A 0.000,B 0.000,C 90.000,E1 11.007} C_DIS
LIN {X -0.156,Y -433.236,Z 706.850,A 0.000,B 0.000,C 90.000,E1 9.029} C_DIS
LIN {X 0.184,Y -436.475,Z 706.837,A 0.000,B 0.000,C 90.000,E1 6.663} C_DIS
LIN {X 0.036,Y -439.280,Z 706.826,A 0.000,B 0.000,C 90.000,E1 4.702} C_DIS
LIN {X 0.123,Y -443.445,Z 706.812,A 0.000,B 0.000,C 90.000,E1 2.064} C_DIS
LIN {X 0.170,Y -447.404,Z 706.799,A 0.000,B 0.000,C 90.000,E1 359.771} C_DIS
LIN {X 0.192,Y -451.093,Z 706.788,A 0.000,B 0.000,C 90.000,E1 357.822} C_DIS
LIN {X 0.042,Y -455.552,Z 706.776,A 0.000,B 0.000,C 90.000,E1 355.584} C_DIS
LIN {X -0.149,Y -459.476,Z 706.765,A 0.000,B 0.000,C 90.000,E1 353.685} C_DIS
LIN {X 0.072,Y -462.721,Z 706.756,A 0.000,B 0.000,C 90.000,E1 352.064} C_DIS
LIN {X 0.163,Y -466.417,Z 706.745,A 0.000,B 0.000,C 90.000,E1 350.151} C_DIS
LIN {X -0.137,Y -468.852,Z 706.738,A 0.000,B 0.000,C 90.000,E1 348.926} C_DIS
LIN {X 0.054,Y -471.127,Z 706.731,A 0.000,B 0.000,C 90.000,E1 347.645} C_DIS
LIN {X 0.150,Y -474.535,Z 706.721,A 0.000,B 0.000,C 90.000,E1 345.755} C_DIS
LIN {X 0.063,Y -476.872,Z 706.714,A 0.000,B 0.000,C 90.000,E1 344.519} C_DIS
LIN {X 0.110,Y -479.813,Z 706.705,A 0.000,B 0.000,C 90.000,E1 342.960} C_DIS
LIN {X 0.059,Y -484.810,Z 706.692,A 0.000,B 0.000,C 90.000,E1 340.496} C_DIS
LIN {X 0.169,Y -489.396,Z 706.680,A 0.000,B 0.000,C 90.000,E1 338.337} C_DIS
LIN {X 0.041,Y -491.034,Z 706.676,A 0.000,B 0.000,C 90.000,E1 337.741} C_DIS
LIN {X 0.051,Y -492.623,Z 706.674,A 0.000,B 0.000,C 90.000,E1 337.283} C_DIS
LIN {X 0.090,Y -493.906,Z 706.672,A 0.000,B 0.000,C 90.000,E1 336.975} C_DIS
LIN {X 0.149,Y -495.986,Z 706.670,A 0.000,B 0.000,C 90.000,E1 336.613} C_DIS
LIN {X -0.003,Y -499.765,Z 706.668,A 0.000,B 0.000,C 90.000,E1 336.177} C_DIS
LIN {X 0.141,Y -504.420,Z 706.665,A 0.000,B 0.000,C 90.000,E1 335.741} C_DIS
LIN {X 0.214,Y -507.458,Z 706.664,A 0.000,B 0.000,C 90.000,E1 335.485} C_DIS
LIN {X 0.150,Y -519.419,Z 706.659,A 0.000,B 0.000,C 90.000,E1 334.665} C_DIS
LIN {X -0.108,Y -525.820,Z 706.657,A 0.000,B 0.000,C 90.000,E1 334.280} C_DIS
LIN {X -0.113,Y -537.888,Z 706.653,A 0.000,B 0.000,C 90.000,E1 333.461} C_DIS
LIN {X 0.245,Y -545.284,Z 706.649,A 0.000,B 0.000,C 90.000,E1 332.871} C_DIS
LIN {X 0.016,Y -551.030,Z 706.647,A 0.000,B 0.000,C 90.000,E1 332.436} C_DIS
LIN {X -0.138,Y -559.263,Z 706.643,A 0.000,B 0.000,C 90.000,E1 331.719} C_DIS
LIN {X 0.187,Y -564.523,Z 706.640,A 0.000,B 0.000,C 90.000,E1 331.179} C_DIS
LIN {X 0.029,Y -570.964,Z 706.636,A 0.000,B 0.000,C 90.000,E1 330.539} C_DIS
LIN {X -0.013,Y -579.652,Z 706.631,A 0.000,B 0.000,C 90.000,E1 329.616} C_DIS
LIN {X 0.116,Y -587.967,Z 706.626,A 0.000,B 0.000,C 90.000,E1 328.663} C_DIS
LIN {X 0.016,Y -596.060,Z 706.621,A 0.000,B 0.000,C 90.000,E1 327.740} C_DIS
LIN {X -0.135,Y -602.660,Z 706.616,A 0.000,B 0.000,C 90.000,E1 326.962} C_DIS
LIN {X 0.083,Y -607.683,Z 706.613,A 0.000,B 0.000,C 90.000,E1 326.294} C_DIS
LIN {X 0.132,Y -614.413,Z 706.608,A 0.000,B 0.000,C 90.000,E1 325.388} C_DIS
LIN {X -0.128,Y -618.058,Z 706.605,A 0.000,B 0.000,C 90.000,E1 324.895} C_DIS
LIN {X -0.023,Y -622.441,Z 706.601,A 0.000,B 0.000,C 90.000,E1 324.242} C_DIS
LIN {X 0.101,Y -628.197,Z 706.596,A 0.000,B 0.000,C 90.000,E1 323.336} C_DIS
LIN {X -0.227,Y -634.245,Z 706.591,A 0.000,B 0.000,C 90.000,E1 322.351} C_DIS
LIN {X 0.301,Y -640.712,Z 706.584,A 0.000,B 0.000,C 90.000,E1 321.170} C_DIS
LIN {X -0.385,Y -645.495,Z 706.580,A 0.000,B 0.000,C 90.000,E1 320.356} C_DIS
LIN {X 0.315,Y -650.707,Z 706.574,A 0.000,B 0.000,C 90.000,E1 319.299} C_DIS
LIN {X -0.320,Y -656.202,Z 706.568,A 0.000,B 0.000,C 90.000,E1 318.243} C_DIS
LIN {X 0.059,Y -659.689,Z 706.564,A 0.000,B 0.000,C 90.000,E1 317.472} C_DIS
LIN {X -0.024,Y -663.975,Z 706.558,A 0.000,B 0.000,C 90.000,E1 316.500} C_DIS
LIN {X -0.030,Y -666.957,Z 706.554,A 0.000,B 0.000,C 90.000,E1 315.769} C_DIS
LIN {X -0.015,Y -671.571,Z 706.548,A 0.000,B 0.000,C 90.000,E1 314.555} C_DIS
LIN {X 0.073,Y -675.011,Z 706.542,A 0.000,B 0.000,C 90.000,E1 313.581} C_DIS
LIN {X 0.223,Y -679.161,Z 706.536,A 0.000,B 0.000,C 90.000,E1 312.366} C_DIS
LIN {X -0.078,Y -682.318,Z 706.530,A 0.000,B 0.000,C 90.000,E1 311.434} C_DIS
LIN {X 0.124,Y -684.521,Z 706.526,A 0.000,B 0.000,C 90.000,E1 310.701} C_DIS
LIN {X -0.117,Y -687.249,Z 706.521,A 0.000,B 0.000,C 90.000,E1 309.769} C_DIS
LIN {X -0.185,Y -690.136,Z 706.514,A 0.000,B 0.000,C 90.000,E1 308.588} C_DIS
LIN {X -0.268,Y -692.079,Z 706.509,A 0.000,B 0.000,C 90.000,E1 307.649} C_DIS
LIN {X 0.230,Y -693.784,Z 706.504,A 0.000,B 0.000,C 90.000,E1 306.664} C_DIS
LIN {X 0.196,Y -695.341,Z 706.499,A 0.000,B 0.000,C 90.000,E1 305.724} C_DIS
LIN {X -0.230,Y -696.653,Z 706.493,A 0.000,B 0.000,C 90.000,E1 304.818} C_DIS
LIN {X -0.060,Y -697.801,Z 706.488,A 0.000,B 0.000,C 90.000,E1 303.865} C_DIS
LIN {X -0.115,Y -698.562,Z 706.484,A 0.000,B 0.000,C 90.000,E1 303.166} C_DIS
LIN {X 0.002,Y -699.824,Z 706.476,A 0.000,B 0.000,C 90.000,E1 301.750} C_DIS
LIN {X 0.213,Y -700.601,Z 706.471,A 0.000,B 0.000,C 90.000,E1 300.797} C_DIS
LIN {X 0.072,Y -701.076,Z 706.466,A 0.000,B 0.000,C 90.000,E1 299.873} C_DIS
LIN {X -0.130,Y -701.523,Z 706.458,A 0.000,B 0.000,C 90.000,E1 298.487} C_DIS
LIN {X -0.383,Y -702.130,Z 706.449,A 0.000,B 0.000,C 90.000,E1 296.873} C_DIS
LIN {X 0.076,Y -702.798,Z 706.443,A 0.000,B 0.000,C 90.000,E1 295.668} C_DIS
LIN {X 0.002,Y -702.896,Z 706.440,A 0.000,B 0.000,C 90.000,E1 295.207} C_DIS
LIN {X -0.015,Y -702.728,Z 706.439,A 0.000,B 0.000,C 90.000,E1 294.975} C_DIS
LIN {X -0.093,Y -702.076,Z 706.436,A 0.000,B 0.000,C 90.000,E1 294.515} C_DIS
LIN {X 0.184,Y -701.153,Z 706.435,A 0.000,B 0.000,C 90.000,E1 294.259} C_DIS
LIN {X -0.332,Y -699.200,Z 706.433,A 0.000,B 0.000,C 90.000,E1 293.951} C_DIS
LIN {X -0.197,Y -698.441,Z 706.432,A 0.000,B 0.000,C 90.000,E1 293.823} C_DIS
LIN {X -0.065,Y -697.491,Z 706.432,A 0.000,B 0.000,C 90.000,E1 293.695} C_DIS
LIN {X 0.066,Y -696.070,Z 706.431,A 0.000,B 0.000,C 90.000,E1 293.567} C_DIS
LIN {X -0.229,Y -689.216,Z 706.429,A 0.000,B 0.000,C 90.000,E1 293.206} C_DIS
LIN {X 0.301,Y -687.130,Z 706.428,A 0.000,B 0.000,C 90.000,E1 293.078} C_DIS
LIN {X 0.320,Y -681.549,Z 706.428,A 0.000,B 0.000,C 90.000,E1 292.950} C_DIS
LIN {X 0.006,Y -677.665,Z 706.427,A 0.000,B 0.000,C 90.000,E1 292.898} C_DIS
LIN {X 0.106,Y -663.598,Z 706.426,A 0.000,B 0.000,C 90.000,E1 292.717} C_DIS
LIN {X 0.174,Y -642.851,Z 706.424,A 0.000,B 0.000,C 90.000,E1 292.386} C_DIS
LIN {X -0.005,Y -633.154,Z 706.423,A 0.000,B 0.000,C 90.000,E1 292.206} C_DIS
LIN {X -0.146,Y -619.816,Z 706.422,A 0.000,B 0.000,C 90.000,E1 291.897} C_DIS
LIN {X -0.209,Y -595.757,Z 706.418,A 0.000,B 0.000,C 90.000,E1 291.227} C_DIS
LIN {X 0.156,Y -574.689,Z 706.414,A 0.000,B 0.000,C 90.000,E1 290.556} C_DIS
LIN {X -0.122,Y -569.119,Z 706.413,A 0.000,B 0.000,C 90.000,E1 290.429} C_DIS
LIN {X -0.157,Y -562.203,Z 706.412,A 0.000,B 0.000,C 90.000,E1 290.174} C_DIS
LIN {X 0.323,Y -559.246,Z 706.411,A 0.000,B 0.000,C 90.000,E1 289.993} C_DIS
LIN {X -0.031,Y -556.110,Z 706.410,A 0.000,B 0.000,C 90.000,E1 289.812} C_DIS
LIN {X -0.064,Y -556.073,Z 706.410,A 0.000,B 0.000,C 90.000,E1 289.812} C_DIS
LIN {X -0.133,Y -555.273,Z 706.409,A 0.000,B 0.000,C 90.000,E1 289.631} C_DIS
LIN {X -0.115,Y -554.636,Z 706.406,A 0.000,B 0.000,C 90.000,E1 289.141} C_DIS
LIN {X -0.009,Y -553.939,Z 706.397,A 0.000,B 0.000,C 90.000,E1 287.457} C_DIS
LIN {X -0.074,Y -553.307,Z 706.388,A 0.000,B 0.000,C 90.000,E1 285.788} C_DIS
LIN {X -0.156,Y -552.729,Z 706.378,A 0.000,B 0.000,C 90.000,E1 284.120} C_DIS
LIN {X 0.140,Y -552.106,Z 706.369,A 0.000,B 0.000,C 90.000,E1 282.411} C_DIS
LIN {X 0.198,Y -551.429,Z 706.360,A 0.000,B 0.000,C 90.000,E1 280.725} C_DIS
LIN {X -0.067,Y -550.352,Z 706.347,A 0.000,B 0.000,C 90.000,E1 278.511} C_DIS
LIN {X -0.088,Y -549.619,Z 706.336,A 0.000,B 0.000,C 90.000,E1 276.549} C_DIS
LIN {X -0.085,Y -549.137,Z 706.324,A 0.000,B 0.000,C 90.000,E1 274.302} C_DIS
LIN {X 0.220,Y -548.810,Z 706.316,A 0.000,B 0.000,C 90.000,E1 272.865} C_DIS
LIN {X -0.016,Y -548.293,Z 706.307,A 0.000,B 0.000,C 90.000,E1 271.203} C_DIS
LIN {X 0.133,Y -547.893,Z 706.302,A 0.000,B 0.000,C 90.000,E1 270.344} C_DIS
LIN {X -0.133,Y -546.841,Z 706.293,A 0.000,B 0.000,C 90.000,E1 268.682} C_DIS
LIN {X 0.132,Y -545.854,Z 706.283,A 0.000,B 0.000,C 90.000,E1 266.963} C_DIS
LIN {X -0.171,Y -544.845,Z 706.275,A 0.000,B 0.000,C 90.000,E1 265.584} C_DIS
LIN {X 0.129,Y -543.633,Z 706.266,A 0.000,B 0.000,C 90.000,E1 263.856} C_DIS
LIN {X -0.227,Y -542.706,Z 706.260,A 0.000,B 0.000,C 90.000,E1 262.761} C_DIS
LIN {X 0.159,Y -540.874,Z 706.249,A 0.000,B 0.000,C 90.000,E1 260.735} C_DIS
LIN {X -0.097,Y -539.582,Z 706.241,A 0.000,B 0.000,C 90.000,E1 259.342} C_DIS
LIN {X -0.142,Y -537.756,Z 706.230,A 0.000,B 0.000,C 90.000,E1 257.353} C_DIS
LIN {X 0.013,Y -535.912,Z 706.219,A 0.000,B 0.000,C 90.000,E1 255.338} C_DIS
LIN {X -0.155,Y -534.805,Z 706.212,A 0.000,B 0.000,C 90.000,E1 254.212} C_DIS
LIN {X -0.153,Y -533.345,Z 706.204,A 0.000,B 0.000,C 90.000,E1 252.779} C_DIS
LIN {X -0.019,Y -531.916,Z 706.196,A 0.000,B 0.000,C 90.000,E1 251.329} C_DIS
LIN {X -0.104,Y -530.662,Z 706.190,A 0.000,B 0.000,C 90.000,E1 250.188} C_DIS
LIN {X 0.150,Y -528.792,Z 706.182,A 0.000,B 0.000,C 90.000,E1 248.720} C_DIS
LIN {X 0.077,Y -526.710,Z 706.174,A 0.000,B 0.000,C 90.000,E1 247.283} C_DIS
LIN {X 0.286,Y -525.052,Z 706.167,A 0.000,B 0.000,C 90.000,E1 246.102} C_DIS
LIN {X -0.174,Y -522.147,Z 706.158,A 0.000,B 0.000,C 90.000,E1 244.409} C_DIS
LIN {X 0.031,Y -520.617,Z 706.153,A 0.000,B 0.000,C 90.000,E1 243.512} C_DIS
LIN {X -0.109,Y -518.414,Z 706.146,A 0.000,B 0.000,C 90.000,E1 242.359} C_DIS
LIN {X 0.071,Y -515.534,Z 706.138,A 0.000,B 0.000,C 90.000,E1 240.873} C_DIS
LIN {X -0.002,Y -512.477,Z 706.130,A 0.000,B 0.000,C 90.000,E1 239.410} C_DIS
LIN {X -0.228,Y -508.705,Z 706.120,A 0.000,B 0.000,C 90.000,E1 237.661} C_DIS
LIN {X 0.123,Y -505.531,Z 706.112,A 0.000,B 0.000,C 90.000,E1 236.135} C_DIS
LIN {X -0.173,Y -502.963,Z 706.105,A 0.000,B 0.000,C 90.000,E1 234.975} C_DIS
LIN {X -0.105,Y -500.973,Z 706.100,A 0.000,B 0.000,C 90.000,E1 234.069} C_DIS
LIN {X 0.109,Y -497.910,Z 706.094,A 0.000,B 0.000,C 90.000,E1 232.844} C_DIS
LIN {X 0.137,Y -494.079,Z 706.085,A 0.000,B 0.000,C 90.000,E1 231.331} C_DIS
LIN {X 0.018,Y -488.898,Z 706.073,A 0.000,B 0.000,C 90.000,E1 229.218} C_DIS
LIN {X -0.014,Y -486.055,Z 706.067,A 0.000,B 0.000,C 90.000,E1 228.000} C_DIS
LIN {X 0.310,Y -481.211,Z 706.055,A 0.000,B 0.000,C 90.000,E1 225.810} C_DIS
LIN {X -0.301,Y -477.099,Z 706.044,A 0.000,B 0.000,C 90.000,E1 224.028} C_DIS
LIN {X -0.089,Y -473.610,Z 706.036,A 0.000,B 0.000,C 90.000,E1 222.447} C_DIS
LIN {X -0.040,Y -470.979,Z 706.029,A 0.000,B 0.000,C 90.000,E1 221.191} C_DIS
LIN {X 0.205,Y -466.976,Z 706.018,A 0.000,B 0.000,C 90.000,E1 219.277} C_DIS
LIN {X -0.045,Y -463.530,Z 706.010,A 0.000,B 0.000,C 90.000,E1 217.729} C_DIS
LIN {X 0.117,Y -459.443,Z 705.999,A 0.000,B 0.000,C 90.000,E1 215.804} C_DIS
LIN {X 0.188,Y -456.387,Z 705.990,A 0.000,B 0.000,C 90.000,E1 214.199} C_DIS
LIN {X -0.241,Y -452.115,Z 705.978,A 0.000,B 0.000,C 90.000,E1 212.005} C_DIS
LIN {X -0.176,Y -447.292,Z 705.963,A 0.000,B 0.000,C 90.000,E1 209.411} C_DIS
LIN {X 0.000,Y -443.793,Z 705.952,A 0.000,B 0.000,C 90.000,E1 207.436} C_DIS
LIN {X 0.074,Y -440.192,Z 705.942,A 0.000,B 0.000,C 90.000,E1 205.463} C_DIS
LIN {X 0.045,Y -437.175,Z 705.932,A 0.000,B 0.000,C 90.000,E1 203.823} C_DIS
LIN {X -0.048,Y -434.790,Z 705.925,A 0.000,B 0.000,C 90.000,E1 202.514} C_DIS
LIN {X 0.261,Y -431.147,Z 705.914,A 0.000,B 0.000,C 90.000,E1 200.482} C_DIS
LIN {X -0.215,Y -427.533,Z 705.903,A 0.000,B 0.000,C 90.000,E1 198.544} C_DIS
LIN {X 0.104,Y -423.249,Z 705.890,A 0.000,B 0.000,C 90.000,E1 196.150} C_DIS
LIN {X 0.187,Y -418.923,Z 705.877,A 0.000,B 0.000,C 90.000,E1 193.772} C_DIS
LIN {X -0.055,Y -414.792,Z 705.863,A 0.000,B 0.000,C 90.000,E1 191.422} C_DIS
LIN {X -0.165,Y -411.883,Z 705.854,A 0.000,B 0.000,C 90.000,E1 189.726} C_DIS
LIN {X 0.001,Y -407.540,Z 705.839,A 0.000,B 0.000,C 90.000,E1 186.947} C_DIS
LIN {X -0.034,Y -404.973,Z 705.829,A 0.000,B 0.000,C 90.000,E1 185.220} C_DIS
LIN {X -0.166,Y -402.011,Z 705.817,A 0.000,B 0.000,C 90.000,E1 183.151} C_DIS
LIN {X -0.156,Y -398.259,Z 705.800,A 0.000,B 0.000,C 90.000,E1 180.000} C_DIS
LIN {X 0.073,Y -394.868,Z 705.780,A 0.000,B 0.000,C 90.000,E1 176.445} C_DIS
LIN {X 0.140,Y -392.163,Z 705.757,A 0.000,B 0.000,C 90.000,E1 172.186} C_DIS
LIN {X -0.134,Y -391.255,Z 705.745,A 0.000,B 0.000,C 90.000,E1 170.095} C_DIS
LIN {X 0.027,Y -390.629,Z 705.733,A 0.000,B 0.000,C 90.000,E1 167.937} C_DIS
LIN {X -0.041,Y -389.980,Z 705.721,A 0.000,B 0.000,C 90.000,E1 165.811} C_DIS
LIN {X -0.089,Y -389.479,Z 705.707,A 0.000,B 0.000,C 90.000,E1 163.323} C_DIS
LIN {X 0.186,Y -389.312,Z 705.693,A 0.000,B 0.000,C 90.000,E1 160.786} C_DIS
LIN {X 0.041,Y -389.277,Z 705.682,A 0.000,B 0.000,C 90.000,E1 158.666} C_DIS
LIN {X -0.013,Y -389.411,Z 705.668,A 0.000,B 0.000,C 90.000,E1 156.177} C_DIS
LIN {X -0.085,Y -389.716,Z 705.654,A 0.000,B 0.000,C 90.000,E1 153.691} C_DIS
LIN {X -0.005,Y -389.936,Z 705.644,A 0.000,B 0.000,C 90.000,E1 151.897} C_DIS
